  //---------------------------------------------------------------------------
  E_PROGRESS.PROGRESS_BUSY:
    _eRslt                      := StationsClearAll(TRUE); // all xts station queues clear
    IF (_eRslt = E_PROGRESS.PROGRESS_DONE)
    THEN
      _eState                   := E_PROGRESS.PROGRESS_PREPARE;
    ELSE
      IF (_eRslt = E_PROGRESS.PROGRESS_ERROR)
      THEN
        _eState                 := E_PROGRESS.PROGRESS_ERROR;
      END_IF
    END_IF

  E_PROGRESS.PROGRESS_PREPARE:
    _eRslt                      := _MoverItf[_nMover].SendToModuloPosCa(TRUE, _stMoveData);

    IF (_eRslt = E_PROGRESS.PROGRESS_ERROR)
    THEN
      _eState                   := E_PROGRESS.PROGRESS_ERROR;
      _nErrorId                 := _MoverInfo[_nMover].nErrorId;
      _eRslt                    := _MoverItf[_nMover].SendToModuloPosCa(FALSE, _stMoveData); 

    ELSIF (_eRslt = E_PROGRESS.PROGRESS_DONE)
    THEN
      _eState                   := E_PROGRESS.PROGRESS_STARTUP;
      _eRslt                    := _MoverItf[_nMover].SendToModuloPosCa(FALSE, _stMoveData);
    END_IF

  //---------------------------------------------------------------------------
  E_PROGRESS.PROGRESS_STARTUP:
    IF (_nMover > GVL_XTS.XpuInfo.nDetectedAxisCount-1)
    THEN
      // all mover are sent to start position, now prepare ticket for Mover 1
      _eState                         := E_PROGRESS.PROGRESS_CHECK;
      // ticket data
      _stMoverDataSend.nMask          := TO_USINT(EXPT(2,_StationStart.nConfiguredStopCount))-1;
      _stMoverDataSend.nMoverId       := TO_USINT(1);
      _stMoverDataSend.nTargetStation := TO_USINT(_nStartStation);
  
      IF (_nStartStation > 0) AND
         (_nStartStation < MAX_STATION+1)
      THEN
        _stListResult           := _ItfStationList[_nStartStation].AddTailValue(_stMoverDataSend); // add first mover to list of _ItfStations[_nStartStation]
      END_IF

    ELSE
      _nMover                   := _nMover + 1;                                                 // increment mover ID
      _stMoveData.rPos          := _StationStart.rPosWait + 2*_MoverItf[_nMover].RailLength;    // all other mover are commanded an extra round, to make sure that mover 1 is always leading the pack
      _eRslt                    := _MoverItf[_nMover].SendToModuloPosCa(FALSE, _stMoveData);
      _eRslt                    := _MoverItf[_nMover].SendToAbsPosCa(FALSE, _stMoveData);
      _eState                   := E_PROGRESS.PROGRESS_PREPARE;                                 // go back and trigger move
    END_IF

  //---------------------------------------------------------------------------
  E_PROGRESS.PROGRESS_CHECK:
    IF (_MoverInfo[1].bMoverInTarget)
    THEN
      IF (_GroupInfo.AllAxesStanding) // wait for all mover standstill
      THEN
        _stMoveData.rPos        := _MoverInfo[1].rAbsTargetPos;                    // Mover1 position to retrigger the movers

        IF (MAX_MOVER > 1)
        THEN
          _nMover               := 2;
          IF (_stMoveData.rPos < _MoverInfo[_nMover].rAbsActPos)
          THEN
            _stMoveData.rPos    := _stMoveData.rPos + _MoverItf[_nMover].RailLength;
          END_IF
          _eState               := E_PROGRESS.PROGRESS_OCCUPIED;
        ELSE
          _eState               := E_PROGRESS.PROGRESS_WORKING;
        END_IF
      END_IF
    END_IF

  //---------------------------------------------------------------------------
  E_PROGRESS.PROGRESS_OCCUPIED:
    _eRslt                      := _MoverItf[_nMover].SendToAbsPosCa(TRUE, _stMoveData); // retrigger

    IF (_eRslt = E_PROGRESS.PROGRESS_ERROR)
    THEN
      _eState                   := E_PROGRESS.PROGRESS_ERROR;
      _nErrorId                 := _MoverInfo[_nMover].nErrorId;
      _eRslt                    := _MoverItf[_nMover].SendToAbsPosCa(FALSE, _stMoveData); 

    ELSIF (_eRslt = E_PROGRESS.PROGRESS_DONE)
    THEN
      _eState                   := E_PROGRESS.PROGRESS_WORKING;
      _eRslt                    := _MoverItf[_nMover].SendToAbsPosCa(FALSE, _stMoveData);

      // write ticket for mover in station list
      _stMoverDataSend.nMask          := TO_USINT(EXPT(2,_StationStart.nConfiguredStopCount))-1;
      _stMoverDataSend.nMoverId       := TO_USINT(_nMover);
      _stMoverDataSend.nTargetStation := TO_USINT(_nStartStation);

      IF (_nStartStation > 0) AND
         (_nStartStation < MAX_STATION+1)
      THEN
        _stListResult                 := _ItfStationList[_nStartStation].AddTailValue(_stMoverDataSend); // enter in list
      END_IF
    END_IF

  //---------------------------------------------------------------------------
  E_PROGRESS.PROGRESS_WORKING:
    IF (_nMover > GVL_XTS.XpuInfo.nDetectedAxisCount-1)
    THEN
      _eState                   := E_PROGRESS.PROGRESS_DONE;

      IF (_eMessageLevel > E_MessageType.eMessageError)
      THEN
        _stMsg.eType            := E_MessageType.eMessageInfo;
        _stMsg.eSubdevice       := e_Subdevice.TransportUnit_General;
        _stMsg.iErrorNumber     := 0;
        _stMsg.sText            := concat( 'State: ', TO_STRING(THIS^._eState));
        _stMsg.sText            := concat(_stMsg.sText, ': ');
        _stMsg.sText            := concat(_stMsg.sText, TO_STRING(_eState));
        f_MessageSet(_stMsg);
      END_IF
    ELSE
      _nMover                   := _nMover + 1;
      IF (_stMoveData.rPos < _MoverInfo[_nMover].rAbsActPos)
      THEN
        _stMoveData.rPos        := _stMoveData.rPos + _MoverItf[_nMover].RailLength;
      END_IF
      _eState                   := E_PROGRESS.PROGRESS_OCCUPIED;
    END_IF
END_CASE
//-----------------------------------------------------------------------------
//-----------------------------------------------------------------------------

TransportStart                  := _eState;
END_METHOD

PROPERTY XpuCtrl : REFERENCE TO ST_XPU_CTRL
SET
_XpuCtrl REF= XpuCtrl;
END_SET
END_PROPERTY

PROPERTY XpuInfo : REFERENCE TO ST_XPU_INFO
SET
_XpuInfo REF= XpuInfo;
END_SET
END_PROPERTY

METHOD XpuInit : E_PROGRESS
VAR_INPUT
  Execute     : BOOL;
END_VAR
VAR_INST
  _nErrorId   : UDINT;
  _eJobReslt,
  _eState     : E_PROGRESS;
END_VAR
//-----------------------------------------------------------------------------
IF NOT Execute 
THEN 
	_eState                       := E_PROGRESS.PROGRESS_INIT; 
END_IF 
//-----------------------------------------------------------------------------
IF NOT Check() 
THEN 
	XpuInit                       := E_PROGRESS.PROGRESS_ERROR; 
	RETURN; 
END_IF
//-----------------------------------------------------------------------------
//-----------------------------------------------------------------------------
CASE _eState
OF
  E_PROGRESS.PROGRESS_INIT:
    IF Execute
    THEN
      _nErrorId                 := 0;
      _XpuCtrl.Cmd              := E_XPU_CTRL.XTS_CMD_NULL; // clear interface

      _eState                   := E_PROGRESS.PROGRESS_BUSY;
    END_IF
  //---------------------------------------------------------------------------
  //---------------------------------------------------------------------------
  E_PROGRESS.PROGRESS_BUSY:
    _XpuCtrl.Cmd                := E_XPU_CTRL.XTS_CMD_INIT; // start Xpu init

    IF (f_GetProgress(_XpuState.State) = E_PROGRESS.PROGRESS_DONE)         // check Xpu init done
    THEN
      _eState                   := E_PROGRESS.PROGRESS_PREPARE;

    ELSIF (f_GetProgress(_XpuState.State) = E_PROGRESS.PROGRESS_ERROR)     // check for error
    THEN
      _eState                   := E_PROGRESS.PROGRESS_ERROR;
    END_IF
  //---------------------------------------------------------------------------
  //---------------------------------------------------------------------------
  E_PROGRESS.PROGRESS_PREPARE:
    _XpuCtrl.Cmd                := E_XPU_CTRL.XTS_IDLE;     // Xpu start cyclic checks and mover detection

    IF (f_GetProgress(_XpuState.State) = E_PROGRESS.PROGRESS_ERROR)     // check for error
    THEN
      _eState                   := E_PROGRESS.PROGRESS_ERROR;

    ELSIF (f_GetProgress(_XpuState.State) = E_PROGRESS.PROGRESS_WORKING)      // check Xpu Idle working
    THEN
      _eState                   := E_PROGRESS.PROGRESS_STARTUP;

    END_IF
  //---------------------------------------------------------------------------
  //---------------------------------------------------------------------------
  E_PROGRESS.PROGRESS_STARTUP:
    IF (f_GetProgress(_XpuState.State) = E_PROGRESS.PROGRESS_ERROR)
    THEN
      _eState                   := E_PROGRESS.PROGRESS_ERROR;

    ELSIF (_XpuState.Check = E_XPU_CHECK.MOVER_ID_SIMULATION) OR
          (_XpuState.Check = E_XPU_CHECK.MOVER_ID_STANDARD)   OR
          (_XpuState.Check = E_XPU_CHECK.MOVER_ID_DETECTION_VALID)
    THEN
      _eState                   := E_PROGRESS.PROGRESS_DONE;

      IF (_eMessageLevel = E_MessageType.eMessageVerbose)
      THEN
        _stMsg.eType            := E_MessageType.eMessageVerbose;
        _stMsg.eSubdevice       := e_Subdevice.TransportUnit_General;
        _stMsg.iErrorNumber     := 0;
        _stMsg.sText            := concat( 'State: ', TO_STRING(THIS^._eState));
        _stMsg.sText            := concat(_stMsg.sText, ': ');
        _stMsg.sText            := concat(_stMsg.sText, TO_STRING(_eState));
        f_MessageSet(_stMsg);
      END_IF
    END_IF
END_CASE
//-----------------------------------------------------------------------------
//-----------------------------------------------------------------------------
XpuInit                         := _eState;
END_METHOD

PROPERTY XpuState : REFERENCE TO ST_XPU_STATE
SET
_XpuState ref= XpuState;
END_SET
END_PROPERTY

END_FUNCTION_BLOCK

// ---- XTS/CaGroup/FB_CaGroup.TcPOU
//---------------------------------------------------------------------------------------------------------------
//
//  HAUD 2023.12.13
//
//
//  fb_CaGroup
//  - handles CA group states
//  - add mover to group
//  - remove mover from group
//  - clear group error
//  - startup procedure for getting group ready to work
//
//
//  VAR INPUT / OUTPUT --> see properties
//
//---------------------------------------------------------------------------------------------------------------//
// This SOFTWARE is provided as an Exemple by THE PROVIDER "as is" and "with all faults." THE PROVIDER makes no  //
// representations or warranties of any kind concerning the safety, suitability, lack of viruses, inaccuracies,  //
// typographical errors, or other harmful components of this SOFTWARE. There are inherent dangers in the use of  //
// any software, and you are solely responsible for determining whether this SOFTWARE is compatible with your    //
// equipment and other software installed on your equipment. You are also solely responsible for the protection  //
// of your equipment and backup of your data, and THE PROVIDER will not be liable for any damages you may suffer //
// in connection with using, modifying, or distributing this SOFTWARE.                                           //
//---------------------------------------------------------------------------------------------------------------//
FUNCTION_BLOCK FB_CaGroup	IMPLEMENTS I_XtsTransport_CaGroup
VAR CONSTANT
{attribute 'hide'} 
  GROUP_HALT_JERK             : LREAL := 500_000.0;
{attribute 'hide'} 
  GROUP_HALT_DEC              : LREAL :=  12_500.0;
END_VAR
VAR
  _eCheck                     : E_GROUP_CHECK;
  _bError                     : BOOL;

  _GroupRef                   : REFERENCE TO Tc3_McCoordinatedMotion.AXES_GROUP_REF;

  _AxisRefMover               : REFERENCE TO ARRAY[1..MAX_MOVER] OF Tc2_MC2.AXIS_REF;
  _MoverItf                   : REFERENCE TO ARRAY[1..MAX_MOVER] OF I_XtsTransport_Mover;  // mover methods

  _stMoveData                 : ST_MOVE_DATA; // dyn constraints for _MoverItf[i].Halt(Execute, stMoveData)

  // CA group fb instances
  _fbAddAxisGroup             : ARRAY[1..MAX_MOVER] OF Tc3_McCoordinatedMotion.MC_AddAxisToGroup;
  _fbRemoveAxisGroup          : ARRAY[1..MAX_MOVER] OF Tc3_McCoordinatedMotion.MC_RemoveAxisFromGroup;

  _fbGroupDisable             : Tc3_McCoordinatedMotion.MC_GroupDisable;
  _fbGroupEnable              : Tc3_McCoordinatedMotion.MC_GroupEnable;
  _fbGroupErrorRead           : Tc3_McCoordinatedMotion.MC_GroupReadError;
  _fbGroupStatusRead          : Tc3_McCoordinatedMotion.MC_GroupReadStatus;
  _fbGroupReset               : Tc3_McCoordinatedMotion.MC_GroupReset;
  _fbGroupStop                : Tc3_McCoordinatedMotion.MC_GroupStop;

  _stGroupInfo                : ST_GROUP_INFO;  // additional bits about the state of the CA group

  _rtrigGroupStatusRead,
  _rtrigGroupErrorRead        : Tc2_Standard.R_TRIG;

  _stMsg                      : ST_Message;
  _eMessageLevel              : E_MessageType;
END_VAR

METHOD AddAll : E_PROGRESS
VAR_INPUT
  Execute     : BOOL;
END_VAR
VAR_INST
  _nErrorId   : UDINT;
  _eState     : E_PROGRESS;

  _nMover     : UINT;
END_VAR
IF NOT Execute THEN _eState     := E_PROGRESS.PROGRESS_INIT; END_IF 
IF NOT Check() THEN AddAll := E_PROGRESS.PROGRESS_ERROR; RETURN; END_IF


CASE _eState
OF
  E_PROGRESS.PROGRESS_INIT:
    IF Execute
    THEN
      _nErrorId               := 0;
      _nMover                 := 1;

      IF (_stGroupInfo.AxisCount < MAX_MOVER)
      THEN
        _eState               := E_PROGRESS.PROGRESS_BUSY;

      ELSE
        _eState               := E_PROGRESS.PROGRESS_DONE;

        IF (_eMessageLevel = E_MessageType.eMessageVerbose)
        THEN
          _stMsg.eType        := E_MessageType.eMessageVerbose;
          _stMsg.eSubdevice   := e_Subdevice.fbGroupAddAxis;
          _stMsg.iErrorNumber := _nMover;
          _stMsg.sText        := TO_STRING(_eState);
          f_MessageSet(_stMsg);
        END_IF
      END_IF
    END_IF
END_CASE
//-----------------------------------------------------------------------------
//-----------------------------------------------------------------------------
CASE _eState
OF
  E_PROGRESS.PROGRESS_BUSY:
    IF (_eMessageLevel = E_MessageType.eMessageVerbose)
    THEN
      _stMsg.eType            := E_MessageType.eMessageVerbose;
      _stMsg.eSubdevice       := e_Subdevice.fbGroupAddAxis;
      _stMsg.iErrorNumber     := _nMover;
      _stMsg.sText            := TO_STRING(_eState);
      f_MessageSet(_stMsg);
    END_IF

    _eState                   := E_PROGRESS.PROGRESS_PREPARE;
    _fbAddAxisGroup[_nMover](
                AxesGroup     := _GroupRef, 
                Axis          := _AxisRefMover[_nMover], 
                Execute       := FALSE, 
                IdentInGroup  := UDINT_TO_IDENTINGROUP(_AxisRefMover[_nMover].NcToPlc.AxisId));
END_CASE
//-----------------------------------------------------------------------------
//-----------------------------------------------------------------------------
CASE _eState
OF
  E_PROGRESS.PROGRESS_PREPARE:
    _fbAddAxisGroup[_nMover](
                AxesGroup     := _GroupRef, 
                Axis          := _AxisRefMover[_nMover], 
                Execute       := TRUE, 
                IdentInGroup  := UDINT_TO_IDENTINGROUP(_AxisRefMover[_nMover].NcToPlc.AxisId));

    IF (_fbAddAxisGroup[_nMover].Error)
    THEN
      _eState                 := E_PROGRESS.PROGRESS_ERROR;
      _nErrorId               := _fbAddAxisGroup[_nMover].ErrorId;

      _stMsg.eType            := E_MessageType.eMessageError;
      _stMsg.eSubdevice       := e_Subdevice.fbGroupAddAxis;
      _stMsg.iErrorNumber     := _nErrorId;
      _stMsg.sText            := TO_STRING(_eState);
      f_MessageSet(_stMsg);

    ELSIF (_fbAddAxisGroup[_nMover].Done)
    THEN
      _eState                 := E_PROGRESS.PROGRESS_CHECK;

      IF (_eMessageLevel = E_MessageType.eMessageVerbose)
      THEN
        _stMsg.eType          := E_MessageType.eMessageVerbose;
        _stMsg.eSubdevice     := e_Subdevice.fbGroupAddAxis;
        _stMsg.iErrorNumber   := _nMover;
        _stMsg.sText          := TO_STRING(_eState);
        f_MessageSet(_stMsg);
      END_IF
    END_IF
END_CASE
//-----------------------------------------------------------------------------
//-----------------------------------------------------------------------------
CASE _eState
OF
  E_PROGRESS.PROGRESS_CHECK:
    _eState                   := E_PROGRESS.PROGRESS_OCCUPIED;
    _fbAddAxisGroup[_nMover](
                AxesGroup     := _GroupRef, 
                Axis          := _AxisRefMover[_nMover], 
                Execute       := FALSE, 
                IdentInGroup  := UDINT_TO_IDENTINGROUP(_AxisRefMover[_nMover].NcToPlc.AxisId));
END_CASE
//-----------------------------------------------------------------------------
//-----------------------------------------------------------------------------
CASE _eState
OF
  E_PROGRESS.PROGRESS_OCCUPIED:
    IF (_nMover > MAX_MOVER-1)
    THEN
      _eState                 := E_PROGRESS.PROGRESS_DONE;

      IF (_eMessageLevel > E_MessageType.eMessageError)
      THEN
        _stMsg.eType          := E_MessageType.eMessageInfo;
        _stMsg.eSubdevice     := e_Subdevice.fbGroupAddAxis;
        _stMsg.iErrorNumber   := MAX_MOVER;
        _stMsg.sText          := TO_STRING(_eState);
        f_MessageSet(_stMsg);
      END_IF
    ELSE
      _nMover                 := _nMover + 1;
      _eState                 := E_PROGRESS.PROGRESS_BUSY;
    END_IF
END_CASE
//-----------------------------------------------------------------------------
//-----------------------------------------------------------------------------

AddAll                   := _eState;
END_METHOD

PROPERTY AxisRef : REFERENCE TO ARRAY[1..MAX_MOVER] OF Tc2_MC2.AXIS_REF
SET
_AxisRefMover REF= AxisRef;
END_SET
END_PROPERTY

METHOD PROTECTED Check : BOOL

IF NOT __ISVALIDREF(_GroupRef)
THEN
  _eCheck                     := E_GROUP_CHECK.CHECK_GROUP_REF_INVALID;
  RETURN;
END_IF

IF NOT __ISVALIDREF(_AxisRefMover)
THEN
  _eCheck                     := E_GROUP_CHECK.CHECK_AXIS_REF_INVALID;
  RETURN;
END_IF

IF NOT __ISVALIDREF(_MoverItf)
THEN
  _eCheck                     := E_GROUP_CHECK.CHECK_Mover_ITF_REF_INVALID;
  RETURN;
END_IF

_eCheck                       := E_GROUP_CHECK.CHECK_DONE;
Check                         := TRUE;
END_METHOD

METHOD Disable : E_PROGRESS
VAR_INPUT
  Execute     : BOOL;
END_VAR
VAR_INST
  _nErrorId   : UDINT;
  _eState     : E_PROGRESS;

  _nMover     : UINT;
END_VAR
IF NOT Execute THEN _eState       := E_PROGRESS.PROGRESS_INIT; END_IF 
IF NOT Check() THEN Disable  := E_PROGRESS.PROGRESS_ERROR; RETURN; END_IF


CASE _eState
OF
  E_PROGRESS.PROGRESS_INIT:
    IF Execute
    THEN
      _nErrorId               := 0;
      _nMover                 := 1;
      _eState                 := E_PROGRESS.PROGRESS_BUSY;
    END_IF
END_CASE
//-----------------------------------------------------------------------------
//-----------------------------------------------------------------------------
CASE _eState
OF
  E_PROGRESS.PROGRESS_BUSY:
    IF (_stGroupInfo.CaGroupState = E_CA_GROUP_STATE.mcGroupStateDisabled)
    THEN
      _eState                 := E_PROGRESS.PROGRESS_DONE;

      IF (_eMessageLevel = E_MessageType.eMessageVerbose)
      THEN
        _stMsg.eType          := E_MessageType.eMessageVerbose;
        _stMsg.eSubdevice     := e_Subdevice.fbGroupDisable;
        _stMsg.iErrorNumber   := _nErrorId;
        _stMsg.sText          := TO_STRING(_eState);
        f_MessageSet(_stMsg);
      END_IF
    ELSE
      _eState                 := E_PROGRESS.PROGRESS_PREPARE;
      _fbGroupDisable(
                AxesGroup     := _GroupRef, 
                Execute       := FALSE);

      _fbGroupReset(
                AxesGroup     := _GroupRef, 
                Execute       := FALSE);
  
      IF (_eMessageLevel = E_MessageType.eMessageVerbose)
      THEN
        _stMsg.eType          := E_MessageType.eMessageVerbose;
        _stMsg.eSubdevice     := e_Subdevice.fbGroupDisable;
        _stMsg.iErrorNumber   := _nErrorId;
        _stMsg.sText          := TO_STRING(_eState);
        f_MessageSet(_stMsg);
      END_IF
    END_IF
END_CASE
//-----------------------------------------------------------------------------
//-----------------------------------------------------------------------------
CASE _eState
OF
  E_PROGRESS.PROGRESS_PREPARE:
    _fbGroupReset(
                AxesGroup     := _GroupRef, 
                Execute       := TRUE);

    IF (_fbGroupReset.Error)
    THEN
      _eState                 := E_PROGRESS.PROGRESS_ERROR;
      _nErrorId               := _fbGroupReset.ErrorId;

      _stMsg.eType            := E_MessageType.eMessageError;
      _stMsg.eSubdevice       := e_Subdevice.fbGroupReset;
      _stMsg.iErrorNumber     := _nErrorId;
      _stMsg.sText            := TO_STRING(_eState);
      f_MessageSet(_stMsg);

      _fbGroupReset(
                AxesGroup     := _GroupRef, 
                Execute       := FALSE);
    ELSE
      IF (_fbGroupReset.Done)
      THEN
        _eState               := E_PROGRESS.PROGRESS_STARTUP;
        _fbGroupReset(
                AxesGroup     := _GroupRef, 
                Execute       := FALSE);
      END_IF
    END_IF
END_CASE
//-----------------------------------------------------------------------------
//-----------------------------------------------------------------------------
CASE _eState
OF
  E_PROGRESS.PROGRESS_STARTUP:
    _fbGroupDisable(
              AxesGroup       := _GroupRef, 
              Execute         := TRUE); 

    IF (_fbGroupDisable.Error)
    THEN
      _eState                 := E_PROGRESS.PROGRESS_ERROR;
      _nErrorId               := _fbGroupDisable.ErrorId;

      _stMsg.eType            := E_MessageType.eMessageError;
      _stMsg.eSubdevice       := e_Subdevice.fbGroupDisable;
      _stMsg.iErrorNumber     := _nErrorId;
      _stMsg.sText            := TO_STRING(_eState);
      f_MessageSet(_stMsg);

      _fbGroupDisable(
              AxesGroup       := _GroupRef, 
              Execute         := FALSE); 


    ELSIF (_fbGroupDisable.Done)
    THEN
      _eState                 := E_PROGRESS.PROGRESS_DONE;

      IF (_eMessageLevel > E_MessageType.eMessageError)
      THEN
        _stMsg.eType          := E_MessageType.eMessageInfo;
        _stMsg.eSubdevice     := e_Subdevice.fbGroupDisable;
        _stMsg.iErrorNumber   := _nErrorId;
        _stMsg.sText          := TO_STRING(_eState);
        f_MessageSet(_stMsg);
      END_IF

      _fbGroupDisable(
              AxesGroup       := _GroupRef, 
              Execute         := FALSE); 
    END_IF
END_CASE
//-----------------------------------------------------------------------------
//-----------------------------------------------------------------------------

Disable                  := _eState;
END_METHOD

METHOD Enable : E_PROGRESS
VAR_INPUT
  Execute     : BOOL;
END_VAR
VAR_INST
  _nErrorId   : UDINT;
  _eState     : E_PROGRESS;

  _nMover     : UINT;
END_VAR
IF NOT Execute THEN _eState       := E_PROGRESS.PROGRESS_INIT; END_IF 
IF NOT Check() THEN Enable   := E_PROGRESS.PROGRESS_ERROR; RETURN; END_IF


CASE _eState
OF
  E_PROGRESS.PROGRESS_INIT:
    IF Execute
    THEN
      _nErrorId               := 0;
      _nMover                 := 1;
      _eState                 := E_PROGRESS.PROGRESS_BUSY;
    END_IF
END_CASE
//-----------------------------------------------------------------------------
//-----------------------------------------------------------------------------
CASE _eState
OF
  E_PROGRESS.PROGRESS_BUSY:
    _eState                   := E_PROGRESS.PROGRESS_PREPARE;
    _fbGroupEnable(
                AxesGroup     := _GroupRef, 
                Execute       := FALSE);

    IF (_eMessageLevel = E_MessageType.eMessageVerbose)
    THEN
      _stMsg.eType            := E_MessageType.eMessageVerbose;
      _stMsg.eSubdevice       := e_Subdevice.fbGroupEnable;
      _stMsg.iErrorNumber     := _nErrorId;
      _stMsg.sText            := TO_STRING(_eState);
      f_MessageSet(_stMsg);
    END_IF
END_CASE
//-----------------------------------------------------------------------------
//-----------------------------------------------------------------------------
CASE _eState
OF
  E_PROGRESS.PROGRESS_PREPARE:
    _fbGroupEnable(
                AxesGroup     := _GroupRef, 
                Execute       := TRUE);

    IF (_fbGroupEnable.Error)
    THEN
      _eState                 := E_PROGRESS.PROGRESS_ERROR;
      _nErrorId               := _fbGroupEnable.ErrorId;

      _stMsg.eType            := E_MessageType.eMessageError;
      _stMsg.eSubdevice       := e_Subdevice.fbGroupEnable;
      _stMsg.iErrorNumber     := _nErrorId;
      _stMsg.sText            := TO_STRING(_eState);
      f_MessageSet(_stMsg);

      _fbGroupEnable(
                AxesGroup     := _GroupRef, 
                Execute       := FALSE);

    ELSIF (_fbGroupEnable.Done)
    THEN
      _eState                 := E_PROGRESS.PROGRESS_DONE;

      IF (_eMessageLevel > E_MessageType.eMessageError)
      THEN
        _stMsg.eType          := E_MessageType.eMessageInfo;
        _stMsg.eSubdevice     := e_Subdevice.fbGroupEnable;
        _stMsg.iErrorNumber   := _nErrorId;
        _stMsg.sText          := TO_STRING(_eState);
        f_MessageSet(_stMsg);
      END_IF
      _fbGroupEnable(
                AxesGroup     := _GroupRef, 
                Execute       := FALSE);
    END_IF
END_CASE
//-----------------------------------------------------------------------------
//-----------------------------------------------------------------------------

Enable                   := _eState;
END_METHOD

PROPERTY GroupInfo : reference to ST_GROUP_INFO
GET
GroupInfo REF= _stGroupInfo;
END_GET
END_PROPERTY

PROPERTY GroupRef : reference to Tc3_McCoordinatedMotion.AXES_GROUP_REF
GET
GroupRef REF= _GroupRef;
END_GET
SET
_GroupRef REF= GroupRef;
END_SET
END_PROPERTY

METHOD InfoCycle : DWORD
VAR_INPUT
  EnableCycle          : BOOL;
END_VAR
VAR_INST
  _nErrorIdADS,
  _nErrorIdRead   : UDINT;

  _nIdx           : udint;
END_VAR
IF NOT Check() THEN RETURN; END_IF

_stMsg.eDevice                              := e_Device.CaGroup;

//-----------------------------------------------------------------------------------------------
// cyclic CA group
//-----------------------------------------------------------------------------------------------
_fbGroupStatusRead(
              AxesGroup                     := _GroupRef, 
              Enable                        := EnableCycle, 
              Valid                         => _stGroupInfo.GroupStatusValid, 
              Busy                          => _stGroupInfo.GroupStatusBusy, 
              GroupMoving                   => _stGroupInfo.GroupMoving, 
              GroupHoming                   => _stGroupInfo.GroupHoming, 
              GroupErrorStop                => _stGroupInfo.GroupErrorStop, 
              GroupNotReady                 => _stGroupInfo.GroupNotReady, 
              GroupStandby                  => _stGroupInfo.GroupStandby, 
              GroupStopping                 => _stGroupInfo.GroupStopping, 
              GroupDisabled                 => _stGroupInfo.GroupDisabled, 
              AllAxesStanding               => _stGroupInfo.AllAxesStanding, 
              ConstantVelocity              => _stGroupInfo.ConstantVelocity, 
              Accelerating                  => _stGroupInfo.Accelerating, 
              Decelerating                  => _stGroupInfo.Decelerating, 
              InPosition                    => _stGroupInfo.InPosition, 
              Error                         => _stGroupInfo.GroupError, 
              ErrorId                       => );

_fbGroupErrorRead(
              AxesGroup                     := _GroupRef, 
              Enable                        := EnableCycle, 
              ErrorId                       => , 
              GroupErrorId                  => _stGroupInfo.GroupErrorId);


_stGroupInfo.AxisCount                      := _GroupRef.NcToPlc.CA.Common.GroupAxesCount;
_stGroupInfo.CaGroupOID                     := _GroupRef.NcToPlc.CA.Common.GroupOID;
_stGroupInfo.CaGroupState                   := TO_UINT(_GroupRef.NcToPlc.CA.Common.GroupStatus.State);

_stGroupInfo.AxisCountEnabled               := 0;
FOR _nIdx := 1 TO MAX_MOVER
DO
  IF (_AxisRefMover[_nIdx].Status.ControlLoopClosed)
  THEN
    _stGroupInfo.AxisCountEnabled           := _stGroupInfo.AxisCountEnabled + 1;
  END_IF
END_FOR	
			  
// fetch internal fb error
_rtrigGroupErrorRead(CLK                    := _fbGroupErrorRead.Error);
IF _rtrigGroupErrorRead.Q
THEN
  _nErrorIdADS                              := _fbGroupErrorRead.ErrorId;

  _stMsg.eType                              := E_MessageType.eMessageError;
  _stMsg.eSubdevice                         := e_Subdevice.fbGroupErrorRead;
  _stMsg.iErrorNumber                       := _nErrorIdADS;
  _stMsg.sText                              := '';
  f_MessageSet(_stMsg);
END_IF

// Dyn constrainst for McHaltAll(method)
_stMoveData.rJerk                           := GROUP_HALT_JERK;
_stMoveData.rAcc                            := GROUP_HALT_DEC;
END_METHOD

METHOD McHaltAll : E_PROGRESS
VAR_INPUT
  Execute       : BOOL;
END_VAR
VAR_INST
  _nErrorId     : UDINT;
  _eState       : E_PROGRESS;
  _eResult      : E_PROGRESS;

  _nMover       : UINT;

  _nRepeat      : UINT;
END_VAR
IF NOT Execute 
THEN 
	_eState     := E_PROGRESS.PROGRESS_INIT; 
END_IF 
IF NOT Check() 
THEN 
	McHaltAll   := E_PROGRESS.PROGRESS_ERROR; 
	RETURN; 
END_IF


CASE _eState
OF
  E_PROGRESS.PROGRESS_INIT:
    IF Execute
    THEN
      _fbGroupStop(
              AxesGroup       := _GroupRef, 
              Execute         := FALSE, 
              Deceleration    := GROUP_HALT_DEC, 
              Jerk            := GROUP_HALT_JERK);

      _nErrorId               := 0;
      _nMover                 := 1;
      _eState                 := E_PROGRESS.PROGRESS_BUSY;
    END_IF
END_CASE

//-----------------------------------------------------------------------------
//-----------------------------------------------------------------------------
CASE _eState
OF
  E_PROGRESS.PROGRESS_BUSY:
    IF NOT (_stGroupInfo.CaGroupState = E_CA_GROUP_STATE.mcGroupStateMoving)
    THEN
      _eState                   := E_PROGRESS.PROGRESS_PREPARE;
    ELSE
      _fbGroupStop(
                AxesGroup       := _GroupRef, 
                Execute         := TRUE, 
                Deceleration    := GROUP_HALT_DEC, 
                Jerk            := GROUP_HALT_JERK);
  
      IF (_fbGroupStop.Error)
      THEN
        _stMsg.eType            := E_MessageType.eMessageError;
        _stMsg.eSubdevice       := e_Subdevice.fbGroupStop;
        _stMsg.iErrorNumber     := _fbGroupStop.ErrorId;
        _stMsg.sText            := TO_STRING(_eState);
        f_MessageSet(_stMsg);
  
        _nRepeat                := _nRepeat + 1;
        _eState                 := E_PROGRESS.PROGRESS_PREPARE;
      ELSE
        IF (_fbGroupStop.Done)
        THEN
          IF (_eMessageLevel = E_MessageType.eMessageVerbose)
          THEN
            _stMsg.eType        := E_MessageType.eMessageVerbose;
            _stMsg.eSubdevice   := e_Subdevice.fbGroupStop;
            _stMsg.iErrorNumber := MAX_MOVER;
            _stMsg.sText        := TO_STRING(_eState);
            f_MessageSet(_stMsg);
          END_IF
          _nRepeat              := 0;
          _eState               := E_PROGRESS.PROGRESS_PREPARE;
        END_IF
      END_IF
    END_IF
END_CASE

//-----------------------------------------------------------------------------
//-----------------------------------------------------------------------------
CASE _eState
OF
  E_PROGRESS.PROGRESS_PREPARE:
    _eState                   := E_PROGRESS.PROGRESS_WORKING;
    _fbGroupStop(
              AxesGroup       := _GroupRef, 
              Execute         := FALSE, 
              Deceleration    := GROUP_HALT_DEC, 
              Jerk            := GROUP_HALT_JERK);

    _eResult                  := _MoverItf[_nMover].Reset(FALSE);
    _eResult                  := _MoverItf[_nMover].Halt(FALSE, _stMoveData);
END_CASE
//-----------------------------------------------------------------------------
//-----------------------------------------------------------------------------
CASE _eState
OF
  E_PROGRESS.PROGRESS_WORKING:
    _eResult                  := _MoverItf[_nMover].Halt(TRUE, _stMoveData);

    IF (_eResult = E_PROGRESS.PROGRESS_DONE)
    THEN
      _eResult                := _MoverItf[_nMover].Halt(FALSE, _stMoveData);
      _eState                 := E_PROGRESS.PROGRESS_STARTUP;

    ELSIF (_eResult = E_PROGRESS.PROGRESS_ERROR)
    THEN
      _nErrorId               := _AxisRefMover[_nMover].NcToPlc.ErrorCode;
      _MoverItf[_nMover].Reset(TRUE);

      _stMsg.eType            := E_MessageType.eMessageError;
      _stMsg.eSubdevice       := e_Subdevice.fbHalt;
      _stMsg.iErrorNumber     := _nErrorId;
      _stMsg.sText            := concat( 'McHaltAll: ', TO_STRING(_eResult));
      _stMsg.sText            := concat(_stMsg.sText, ' MoverId: ');
      _stMsg.sText            := concat(_stMsg.sText, TO_STRING(_nMover));
      f_MessageSet(_stMsg);

      _eState                 := E_PROGRESS.PROGRESS_PREPARE;
    END_IF
END_CASE

//-----------------------------------------------------------------------------
//-----------------------------------------------------------------------------
CASE _eState
OF
  E_PROGRESS.PROGRESS_STARTUP:
    IF (_nMover > MAX_MOVER-1)
    THEN
      _eState                 := E_PROGRESS.PROGRESS_CHECK;
    ELSE
      _nMover                 := _nMover + 1;
      _eState                 := E_PROGRESS.PROGRESS_PREPARE;
    END_IF
END_CASE

//-----------------------------------------------------------------------------
//-----------------------------------------------------------------------------
CASE _eState
OF
  E_PROGRESS.PROGRESS_CHECK:
    _eState                   := E_PROGRESS.PROGRESS_DONE;

    IF (_eMessageLevel > E_MessageType.eMessageError)
    THEN
      _stMsg.eType            := E_MessageType.eMessageInfo;
      _stMsg.eSubdevice       := e_Subdevice.fbCaGroup;
      _stMsg.iErrorNumber     := MAX_MOVER;
      _stMsg.sText            := concat('McHaltAll: ', TO_STRING(_eState));
      f_MessageSet(_stMsg);
    END_IF
END_CASE
//-----------------------------------------------------------------------------
//-----------------------------------------------------------------------------
McHaltAll                     := _eState;
END_METHOD

METHOD McResetAll : E_PROGRESS
VAR_INPUT
  Execute       : BOOL;
END_VAR
VAR_INST
  _nErrorId     : UDINT;
  _eRslt,
  _eState       : E_PROGRESS;

  _nMover       : UINT;
END_VAR
IF NOT Execute THEN _eState     := E_PROGRESS.PROGRESS_INIT; END_IF 
IF NOT Check() THEN McResetAll  := E_PROGRESS.PROGRESS_ERROR; RETURN; END_IF


//-----------------------------------------------------------------------------
//-----------------------------------------------------------------------------
CASE _eState
OF
  E_PROGRESS.PROGRESS_INIT:
    IF Execute
    THEN
      _nErrorId                 := 0;
      _nMover                   := 1;

      _eState                   := E_PROGRESS.PROGRESS_BUSY;
    END_IF
END_CASE
//-----------------------------------------------------------------------------
//-----------------------------------------------------------------------------
CASE _eState
OF
  E_PROGRESS.PROGRESS_BUSY:
    _eState                     := E_PROGRESS.PROGRESS_PREPARE;
    _eRslt                      := _MoverItf[_nMover].Reset(FALSE);
END_CASE
//-----------------------------------------------------------------------------
//-----------------------------------------------------------------------------
CASE _eState
OF
  E_PROGRESS.PROGRESS_PREPARE:
    _eRslt                      := _MoverItf[_nMover].Reset(TRUE);

    IF (_eRslt = E_PROGRESS.PROGRESS_ERROR)
    THEN
      _eState                   := E_PROGRESS.PROGRESS_BUSY;

    ELSIF (_eRslt = E_PROGRESS.PROGRESS_DONE)
    THEN
      _eState                   := E_PROGRESS.PROGRESS_STARTUP;
    END_IF
END_CASE
//-----------------------------------------------------------------------------
//-----------------------------------------------------------------------------
CASE _eState
OF
  E_PROGRESS.PROGRESS_STARTUP:
    _eState                     := E_PROGRESS.PROGRESS_CHECK;
    _eRslt                      := _MoverItf[_nMover].Reset(FALSE);
END_CASE
//-----------------------------------------------------------------------------
//-----------------------------------------------------------------------------
CASE _eState
OF
  E_PROGRESS.PROGRESS_CHECK:
    IF (_nMover > MAX_MOVER-1)
    THEN
      _eState                   := E_PROGRESS.PROGRESS_DONE;

      IF (_eMessageLevel = E_MessageType.eMessageVerbose)
      THEN
        _stMsg.eType            := E_MessageType.eMessageVerbose;
        _stMsg.eSubdevice       := e_Subdevice.fbReset;
        _stMsg.iErrorNumber     := 0;
        _stMsg.sText            := concat( 'State: ', TO_STRING(_eState));
        f_MessageSet(_stMsg);
      END_IF
    ELSE
      _nMover                   := _nMover + 1;
      _eState                   := E_PROGRESS.PROGRESS_BUSY;
    END_IF
END_CASE
//-----------------------------------------------------------------------------
//-----------------------------------------------------------------------------


McResetAll                      := _eState;
END_METHOD

PROPERTY MessageLevel : e_messagetype
SET
_eMessageLevel := MessageLevel;
END_SET
END_PROPERTY

PROPERTY MoverItf : reference TO ARRAY[1..MAX_MOVER] OF I_XtsTransport_Mover
SET
_MoverItf REF= MoverItf;
END_SET
END_PROPERTY

METHOD RemoveAll : E_PROGRESS
VAR_INPUT
  Execute     : BOOL;
END_VAR
VAR_INST
  _nErrorId   : UDINT;
  _eState     : E_PROGRESS;

  _nMover     : UINT;
END_VAR
IF NOT Execute THEN _eState         := E_PROGRESS.PROGRESS_INIT; END_IF 
IF NOT Check() THEN RemoveAll  := E_PROGRESS.PROGRESS_ERROR; RETURN; END_IF


CASE _eState
OF
  E_PROGRESS.PROGRESS_INIT:
    IF Execute
    THEN
      _nErrorId               := 0;
      _nMover                 := 1;

      IF (_stGroupInfo.AxisCount > 0)
      THEN
        _eState               := E_PROGRESS.PROGRESS_BUSY;
      ELSE
        _eState               := E_PROGRESS.PROGRESS_DONE;

        IF (_eMessageLevel = E_MessageType.eMessageVerbose)
        THEN
          _stMsg.eType        := E_MessageType.eMessageVerbose;
          _stMsg.eSubdevice   := e_Subdevice.fbGroupRemoveAxis;
          _stMsg.iErrorNumber := _stGroupInfo.AxisCount;
          _stMsg.sText        := TO_STRING(_eState);
          f_MessageSet(_stMsg);
        END_IF
      END_IF
    END_IF
END_CASE
//-----------------------------------------------------------------------------
//-----------------------------------------------------------------------------
CASE _eState
OF
  E_PROGRESS.PROGRESS_BUSY:
    IF (_eMessageLevel = E_MessageType.eMessageVerbose)
    THEN
      _stMsg.eType          := E_MessageType.eMessageVerbose;
      _stMsg.eSubdevice     := e_Subdevice.fbGroupRemoveAxis;
      _stMsg.iErrorNumber   := _nMover;
      _stMsg.sText          := TO_STRING(_eState);
      //f_MessageSet(_stMsg);
    END_IF

    _eState                 := E_PROGRESS.PROGRESS_PREPARE;
    _fbRemoveAxisGroup[_nMover](
            AxesGroup       := _GroupRef, 
            Execute         := FALSE,
            IdentInGroup    := UDINT_TO_IDENTINGROUP(_AxisRefMover[_nMover].NcToPlc.AxisId));
END_CASE
//-----------------------------------------------------------------------------
//-----------------------------------------------------------------------------
CASE _eState
OF
  E_PROGRESS.PROGRESS_PREPARE:
    _fbRemoveAxisGroup[_nMover](
              AxesGroup       := _GroupRef, 
              Execute         := TRUE,
              IdentInGroup    := UDINT_TO_IDENTINGROUP(_AxisRefMover[_nMover].NcToPlc.AxisId));

    IF (_fbRemoveAxisGroup[_nMover].Error)
    THEN
      _eState                 := E_PROGRESS.PROGRESS_ERROR;
      _nErrorId               := _fbRemoveAxisGroup[_nMover].ErrorId;

      _stMsg.eType            := E_MessageType.eMessageError;
      _stMsg.eSubdevice       := e_Subdevice.fbGroupRemoveAxis;
      _stMsg.iErrorNumber     := _nErrorId;
      _stMsg.sText            := TO_STRING(_eState);
      f_MessageSet(_stMsg);

    ELSIF (_fbRemoveAxisGroup[_nMover].Done)
    THEN
      _eState                 := E_PROGRESS.PROGRESS_CHECK;

      IF (_eMessageLevel = E_MessageType.eMessageVerbose)
      THEN
        _stMsg.eType          := E_MessageType.eMessageVerbose;
        _stMsg.eSubdevice     := e_Subdevice.fbGroupRemoveAxis;
        _stMsg.iErrorNumber   := _nMover;
        _stMsg.sText          := TO_STRING('DONE');
        //f_MessageSet(_stMsg);
      END_IF
    END_IF
END_CASE
//-----------------------------------------------------------------------------
//-----------------------------------------------------------------------------
CASE _eState
OF
  E_PROGRESS.PROGRESS_CHECK:
    _eState                   := E_PROGRESS.PROGRESS_OCCUPIED;
    _fbRemoveAxisGroup[_nMover](
              AxesGroup       := _GroupRef, 
              Execute         := FALSE,
              IdentInGroup    := UDINT_TO_IDENTINGROUP(_AxisRefMover[_nMover].NcToPlc.AxisId));
END_CASE
//-----------------------------------------------------------------------------
//-----------------------------------------------------------------------------
CASE _eState
OF
  E_PROGRESS.PROGRESS_OCCUPIED:
    IF (_nMover > MAX_MOVER-1)
    THEN
      _eState                 := E_PROGRESS.PROGRESS_DONE;

      IF (_eMessageLevel > E_MessageType.eMessageError)
      THEN
        _stMsg.eType          := E_MessageType.eMessageInfo;
        _stMsg.eSubdevice     := e_Subdevice.fbGroupRemoveAxis;
        _stMsg.iErrorNumber   := MAX_MOVER;
        _stMsg.sText          := TO_STRING(_eState);
        f_MessageSet(_stMsg);
      END_IF
    ELSE
      _nMover                 := _nMover + 1;
      _eState                 := E_PROGRESS.PROGRESS_BUSY;
    END_IF
END_CASE
//-----------------------------------------------------------------------------
//-----------------------------------------------------------------------------

RemoveAll                := _eState;
END_METHOD

METHOD Reset : E_PROGRESS
VAR_INPUT
  Execute     : BOOL;
END_VAR
VAR_INST
  _nErrorId   : UDINT;
  _eState     : E_PROGRESS;

  _nMover     : UINT;
END_VAR
IF NOT Execute 
THEN 
	_eState := E_PROGRESS.PROGRESS_INIT; 
END_IF 
IF NOT Check() 
THEN 
	Reset := E_PROGRESS.PROGRESS_ERROR; 
	RETURN; 
END_IF


CASE _eState
OF
  E_PROGRESS.PROGRESS_INIT:
    IF Execute
    THEN
      _nErrorId                 := 0;
      _nMover                   := 1;
      _stGroupInfo.GroupErrorId := 0;
      _stGroupInfo.GroupError   := FALSE;

      _eState                   := E_PROGRESS.PROGRESS_BUSY;
    END_IF
END_CASE
//-----------------------------------------------------------------------------
//-----------------------------------------------------------------------------
CASE _eState
OF
  E_PROGRESS.PROGRESS_BUSY:
    _eState                     := E_PROGRESS.PROGRESS_PREPARE;
    _fbGroupReset(
              AxesGroup         := _GroupRef, 
              Execute           := FALSE);

    IF (_eMessageLevel = E_MessageType.eMessageVerbose)
    THEN
      _stMsg.eType              := E_MessageType.eMessageVerbose;
      _stMsg.eSubdevice         := e_Subdevice.fbGroupReset;
      _stMsg.iErrorNumber       := 0;
      _stMsg.sText              := TO_STRING(_eState);
      //f_MessageSet(_stMsg);
    END_IF
END_CASE
//-----------------------------------------------------------------------------
//-----------------------------------------------------------------------------
CASE _eState
OF
  E_PROGRESS.PROGRESS_PREPARE:
    _fbGroupReset(
              AxesGroup         := _GroupRef, 
              Execute           := TRUE);

    IF (_fbGroupReset.Error)
    THEN
      _eState                   := E_PROGRESS.PROGRESS_ERROR;
      _nErrorId                 := _fbGroupReset.ErrorId;

      _stMsg.eType              := E_MessageType.eMessageError;
      _stMsg.eSubdevice         := e_Subdevice.fbGroupReset;
      _stMsg.iErrorNumber       := _nErrorId;
      _stMsg.sText              := TO_STRING(_eState);
      f_MessageSet(_stMsg);

      _fbGroupReset(
              AxesGroup         := _GroupRef, 
              Execute           := FALSE); 

    ELSIF (_fbGroupReset.Done)
    THEN
      _eState                   := E_PROGRESS.PROGRESS_DONE;

      IF (_eMessageLevel > E_MessageType.eMessageError)
      THEN
        _stMsg.eType            := E_MessageType.eMessageInfo;
        _stMsg.eSubdevice       := e_Subdevice.fbGroupReset;
        _stMsg.iErrorNumber     := _nErrorId;
        _stMsg.sText            := TO_STRING(_eState);
        f_MessageSet(_stMsg);
      END_IF

      _fbGroupReset(
              AxesGroup         := _GroupRef, 
              Execute           := FALSE); 
    END_IF
END_CASE
//-----------------------------------------------------------------------------
//-----------------------------------------------------------------------------

Reset                           := _eState;
END_METHOD

METHOD Stop : E_PROGRESS
VAR_INPUT
  Execute     : BOOL;
END_VAR
VAR_INST
  _nErrorId   : UDINT;
  _eState     : E_PROGRESS;

  _nMover     : UINT;
  _nRepeat    : uint;
END_VAR
IF NOT Execute 
THEN 
	_eState := E_PROGRESS.PROGRESS_INIT; 
END_IF 
IF NOT Check() 
THEN 
	Stop := E_PROGRESS.PROGRESS_ERROR; 
	RETURN; 
END_IF


CASE _eState
OF
  E_PROGRESS.PROGRESS_INIT:
    IF Execute
    THEN
      _nRepeat                  := 0;
      _nErrorId                 := 0;
      _nMover                   := 1;
      _eState                   := E_PROGRESS.PROGRESS_BUSY;
    END_IF
END_CASE
//-----------------------------------------------------------------------------
//-----------------------------------------------------------------------------
CASE _eState
OF
  E_PROGRESS.PROGRESS_BUSY:
    _eState                     := E_PROGRESS.PROGRESS_PREPARE;
    _fbGroupStop(
                AxesGroup       := _GroupRef, 
                Execute         := FALSE, 
                Deceleration    := GROUP_HALT_DEC, 
                Jerk            := GROUP_HALT_JERK);

    IF (_eMessageLevel = E_MessageType.eMessageVerbose)
    THEN
      _stMsg.eType              := E_MessageType.eMessageVerbose;
      _stMsg.eSubdevice         := e_Subdevice.fbGroupStop;
      _stMsg.iErrorNumber       := 0;
      _stMsg.sText              := TO_STRING(_eState);
      f_MessageSet(_stMsg);
    END_IF
END_CASE
//-----------------------------------------------------------------------------
//-----------------------------------------------------------------------------
CASE _eState
OF
  E_PROGRESS.PROGRESS_PREPARE:
    _fbGroupStop(
                AxesGroup       := _GroupRef, 
                Execute         := TRUE, 
                Deceleration    := GROUP_HALT_DEC, 
                Jerk            := GROUP_HALT_JERK);

    IF (_fbGroupStop.Error)
    THEN
      _eState                   := E_PROGRESS.PROGRESS_STARTUP;
      _nErrorId                 := _fbGroupStop.ErrorId;

      _stMsg.eType              := E_MessageType.eMessageError;
      _stMsg.eSubdevice         := e_Subdevice.fbGroupStop;
      _stMsg.iErrorNumber       := _nErrorId;
      _stMsg.sText              := TO_STRING(_eState);
      f_MessageSet(_stMsg);

      _fbGroupReset(
              AxesGroup         := _GroupRef, 
              Execute           := FALSE); 

    ELSIF (_fbGroupStop.Done)
    THEN
      _eState                   := E_PROGRESS.PROGRESS_DONE;

      IF (_eMessageLevel > E_MessageType.eMessageError)
      THEN
        _stMsg.eType            := E_MessageType.eMessageInfo;
        _stMsg.eSubdevice       := e_Subdevice.fbGroupStop;
        _stMsg.iErrorNumber     := _nErrorId;
        _stMsg.sText            := TO_STRING(_eState);
        f_MessageSet(_stMsg);
      END_IF

      _fbGroupStop(
                AxesGroup       := _GroupRef, 
                Execute         := FALSE, 
                Deceleration    := GROUP_HALT_DEC, 
                Jerk            := GROUP_HALT_JERK);
    END_IF
END_CASE
//-----------------------------------------------------------------------------
//-----------------------------------------------------------------------------
CASE _eState
OF
  E_PROGRESS.PROGRESS_STARTUP:
    _fbGroupReset(
              AxesGroup         := _GroupRef, 
              Execute           := TRUE);

    IF (_fbGroupReset.Error)
    THEN
      _nRepeat                  := _nRepeat + 1;
      IF (_nRepeat > 2)
      THEN
        _eState                 := E_PROGRESS.PROGRESS_ERROR;
      END_IF
      _nErrorId                 := _fbGroupReset.ErrorId;

      _stMsg.eType              := E_MessageType.eMessageError;
      _stMsg.eSubdevice         := e_Subdevice.fbGroupStop;
      _stMsg.iErrorNumber       := _nErrorId;
      _stMsg.sText              := TO_STRING(_eState);
      f_MessageSet(_stMsg);

      _fbGroupReset(
              AxesGroup         := _GroupRef, 
              Execute           := FALSE); 

    ELSIF (_fbGroupReset.Done)
    THEN
      _eState                   := E_PROGRESS.PROGRESS_BUSY;

      IF (_eMessageLevel > E_MessageType.eMessageError)
      THEN
        _stMsg.eType            := E_MessageType.eMessageInfo;
        _stMsg.eSubdevice       := e_Subdevice.fbGroupStop;
        _stMsg.iErrorNumber     := _nErrorId;
        _stMsg.sText            := TO_STRING(_eState);
        f_MessageSet(_stMsg);
      END_IF

      _fbGroupReset(
              AxesGroup         := _GroupRef, 
              Execute           := FALSE); 
    END_IF
END_CASE
//-----------------------------------------------------------------------------
//-----------------------------------------------------------------------------

Stop                            := _eState;
END_METHOD

END_FUNCTION_BLOCK

// ---- XTS/Mover/fb_MoverCtrl.TcPOU
//---------------------------------------------------------------------------------------------------------------
//
//  HAUD 2023.12.18
//
//  - XTS_TRANSPORT_LAYER
//
//  fb_MoverCtrl
//  - accepts orders (E_MOVER_CTRL) via cyclic struct interface to execute
//  - interface struct  to extern control
//
//
//---------------------------------------------------------------------------------------------------------------
// This SOFTWARE is provided as an Exemple by THE PROVIDER "as is" and "with all faults." THE PROVIDER makes no 
// representations or warranties of any kind concerning the safety, suitability, lack of viruses, inaccuracies, 
// typographical errors, or other harmful components of this SOFTWARE. There are inherent dangers in the use of 
// any software, and you are solely responsible for determining whether this SOFTWARE is compatible with your 
// equipment and other software installed on your equipment. You are also solely responsible for the protection 
// of your equipment and backup of your data, and THE PROVIDER will not be liable for any damages you may suffer 
// in connection with using, modifying, or distributing this SOFTWARE.
//---------------------------------------------------------------------------------------------------------------
FUNCTION_BLOCK fb_MoverCtrl EXTENDS fb_Mover
VAR
  // Ctrl and State for executing commands
  _stCtrl           : REFERENCE TO ARRAY[1..MAX_MOVER] OF ST_MOVER_CTRL;
  _stState          : REFERENCE TO ARRAY[1..MAX_MOVER] OF ST_MOVER_STATE;

  // data structures to use with commands
  _stMoveData       : REFERENCE TO ARRAY[1..MAX_MOVER] OF ST_MOVE_DATA;
  _stGearData       : REFERENCE TO ARRAY[1..MAX_MOVER] OF ST_GEAR_DATA;

  _eCmd,
  _eCmdOld          : E_MOVER_CTRL;

  _eState           : E_MOVER_STATE;

  _eResult          : E_PROGRESS;
END_VAR

IF NOT Check() THEN RETURN; END_IF

_stMsg.eDevice                := e_Device.Mover + _nMoverId;

// copy to local for debug
_eCmd                         := _stCtrl[_nMoverId].Cmd;

// cyclic check for command change
// get state for cmd
IF (_eCmd <> _eCmdOld)
THEN
  // get matching sdtate for Ctrl.Cmd
  _eState                     := Cmd(_eCmd);
  _eCmdOld                    := _eCmd;
END_IF


CASE _eResult
OF
  E_PROGRESS.PROGRESS_INVALID:
    _stState[_nMoverId].State := E_MOVER_STATE.MOVER_NULL;

  E_PROGRESS.PROGRESS_ERROR:
    _stState[_nMoverId].State := _eState + E_PROGRESS.PROGRESS_ERROR;

  E_PROGRESS.PROGRESS_DONE:
    _stInfo.nErrorId          := 0;
    _stInfo.bMoverError       := FALSE;
    _stState[_nMoverId].State := _eState + E_PROGRESS.PROGRESS_DONE;

ELSE
  // work in progress
  // update progress for extern use
  _stState[_nMoverId].State   := _eState + _eResult;

  CASE _eState
  OF
    E_MOVER_STATE.MOVER_ENABLE:
      _eResult                := Enable(TRUE);
  
    E_MOVER_STATE.MOVER_DISABLE:
      _eResult                := Disable(TRUE);
  
    E_MOVER_STATE.MOVER_MOVE_TO_POS:
      _eResult                := MoveToPos(TRUE, _stMoveData[_nMoverId]);
  
    E_MOVER_STATE.MOVER_MOVE_TO_POS_CA:
      _eResult                := MoveToPosCa(TRUE, _stMoveData[_nMoverId]);
  
    E_MOVER_STATE.MOVER_SEND_TO_POS_CA:
      _eResult                := SendToModuloPosCa(TRUE, _stMoveData[_nMoverId]);
  
    E_MOVER_STATE.MOVER_HALT:
      _eResult                := Halt(TRUE, _stMoveData[_nMoverId]);
  
    E_MOVER_STATE.MOVER_GEAR_IN:
      _eResult                := GearIn(TRUE, _stMoveData[_nMoverId], _stGearData[_nMoverId]);
  
    E_MOVER_STATE.MOVER_GEAR_IN_POS_CA:
      _eResult                := GearInPosCa(TRUE, _stMoveData[_nMoverId], _stGearData[_nMoverId]);
  
    E_MOVER_STATE.MOVER_GEAR_OUT:
      _eResult                := GearOut(TRUE);
  
    E_MOVER_STATE.MOVER_RESET:
      _eResult                := Reset(TRUE);
  ELSE
      _eResult                := E_PROGRESS.PROGRESS_INVALID;
  END_CASE
END_CASE

METHOD PRIVATE Check : BOOL

// The thing that should not be

IF NOT (_nMoverId > 0)
THEN
  _sState                     := 'Mover: missing ID';
  RETURN;
END_IF

IF NOT __ISVALIDREF(_stCtrl)
THEN
  _sState                     := 'Ctrl: missing pointer';
  RETURN;
END_IF

IF NOT __ISVALIDREF(_stState)
THEN
  _sState                     := 'State: missing pointer';
  RETURN;
END_IF

IF NOT __ISVALIDREF(_Mover)
THEN
  _sState                     := 'Mover: missing pointer';
  RETURN;
END_IF

IF NOT __ISVALIDREF(_rLastPosition)
THEN
  _sState                     := '_rLastPosition: missing pointer';
  RETURN;
END_IF

IF NOT __ISVALIDREF(_rLastGap)
THEN
  _sState                     := '_rLastGap: missing pointer';
  RETURN;
END_IF

IF NOT __ISVALIDREF(_stInfo)
THEN
  _sState                     := '_stInfo: missing pointer';
  RETURN;
END_IF

IF NOT __ISVALIDREF(_stGearData)
THEN
  _sState                     := '_stGearData: missing pointer';
  RETURN;
END_IF

IF NOT __ISVALIDREF(_stMoveData)
THEN
  _sState                     := '_stMoveData: missing pointer';
  RETURN;
END_IF

_sState                       := 'CHECK_DONE';
Check                         := TRUE;
END_METHOD

METHOD PRIVATE Cmd : E_MOVER_STATE
VAR_INPUT
  Ctrl      : E_MOVER_CTRL;
END_VAR
VAR_INST
  _eState   : E_MOVER_STATE;
END_VAR
IF NOT Check() THEN Cmd := E_MOVER_STATE.MOVER_NULL;  RETURN; END_IF


CASE Ctrl
OF
  E_MOVER_CTRL.MOVER_ENABLE:
    _eResult          := Enable(FALSE);
    _eState           := E_MOVER_STATE.MOVER_ENABLE;

  E_MOVER_CTRL.MOVER_DISABLE:
    _eResult          := Disable(FALSE);
    _eState           := E_MOVER_STATE.MOVER_DISABLE;

  E_MOVER_CTRL.MOVER_MOVE_TO_POS:
    _eResult          := MoveToPos(FALSE, _stMoveData[_nMoverId]);
    _eState           := E_MOVER_STATE.MOVER_MOVE_TO_POS;

  E_MOVER_CTRL.MOVER_MOVE_TO_POS_CA:
    _eResult          := MoveToPosCa(FALSE, _stMoveData[_nMoverId]);
    _eState           := E_MOVER_STATE.MOVER_MOVE_TO_POS_CA;

  E_MOVER_CTRL.MOVER_SEND_TO_POS_CA:
    _eResult          := SendToModuloPosCa(FALSE, _stMoveData[_nMoverId]);
    _eState           := E_MOVER_STATE.MOVER_SEND_TO_POS_CA;

  E_MOVER_CTRL.MOVER_HALT:
    _eResult          := Halt(FALSE, _stMoveData[_nMoverId]);
    _eState           := E_MOVER_STATE.MOVER_HALT;

  E_MOVER_CTRL.MOVER_GEAR_IN:
    _eResult          := GearIn(FALSE,  _stMoveData[_nMoverId], _stGearData[_nMoverId]);
    _eState           := E_MOVER_STATE.MOVER_GEAR_IN;

  E_MOVER_CTRL.MOVER_GEAR_IN_POS_CA:
    _eResult          := GearInPosCa(FALSE, _stMoveData[_nMoverId], _stGearData[_nMoverId]);
    _eState           := E_MOVER_STATE.MOVER_GEAR_IN_POS_CA;

  E_MOVER_CTRL.MOVER_GEAR_OUT:
    _eResult          := GearOut(FALSE);
    _eState           := E_MOVER_STATE.MOVER_GEAR_OUT;

  E_MOVER_CTRL.MOVER_RESET:
    _eResult          := Reset(FALSE);
    _eState           := E_MOVER_STATE.MOVER_RESET;

ELSE
    _eResult          := E_PROGRESS.PROGRESS_INVALID; 
    _eState           := E_MOVER_STATE.MOVER_NULL;
END_CASE

Cmd                   := _eState;
END_METHOD

PROPERTY Ctrl : REFERENCE TO ARRAY[1..MAX_MOVER] OF ST_MOVER_CTRL
SET
_stCtrl ref= Ctrl;
END_SET
END_PROPERTY

PROPERTY GearData : reference TO ARRAY[1..MAX_MOVER] OF ST_GEAR_DATA
SET
_stGearData REF= GearData;
END_SET
END_PROPERTY

PROPERTY MoveData : reference TO ARRAY[1..MAX_MOVER] OF st_move_data
SET
_stMoveData REF= MoveData;
END_SET
END_PROPERTY

PROPERTY State : REFERENCE TO ARRAY[1..MAX_MOVER] OF ST_MOVER_STATE
SET
_stState ref= State;
END_SET
END_PROPERTY

END_FUNCTION_BLOCK

// ---- XTS/Mover/fb_Mover.TcPOU
//---------------------------------------------------------------------------------------------------------------
//
//  HAUD 2023.12.19
//
//  - XTS_TRANSPORT_LAYER
//
//  fb_Mover
//  - all positioning input is modulo value
//  - wrap MC function blocks
//
//
//---------------------------------------------------------------------------------------------------------------
// This SOFTWARE is provided as an Example by THE PROVIDER "as is" and "with all faults." THE PROVIDER makes no 
// representations or warranties of any kind concerning the safety, suitability, lack of viruses, inaccuracies, 
// typographical errors, or other harmful components of this SOFTWARE. There are inherent dangers in the use of 
// any software, and you are solely responsible for determining whether this SOFTWARE is compatible with your 
// equipment and other software installed on your equipment. You are also solely responsible for the protection 
// of your equipment and backup of your data, and THE PROVIDER will not be liable for any damages you may suffer 
// in connection with using, modifying, or distributing this SOFTWARE.
//---------------------------------------------------------------------------------------------------------------
FUNCTION_BLOCK fb_Mover IMPLEMENTS I_XtsTransport_Mover
VAR
  _nMoverId         : UINT;

  _sState           : STRING;

  _Master,
  _Mover            : REFERENCE TO AXIS_REF;
  _rLastPosition    : REFERENCE TO LREAL;
  _rLastGap         : REFERENCE TO LREAL;

  _RailLength       : LREAL;
  _nSyncStrategy    : Tc3_Mc3Definitions.MC_SYNC_STRATEGY := Tc3_Mc3Definitions.MC_SYNC_STRATEGY.mcSyncStrategySlow; // minimal movement with this strategy 

  // mover compact axis information
  _stInfo           : REFERENCE TO ST_MOVER_INFO; // ActPos, Enable, ...

  _bError           : BOOL;   // used in Cycle()
  _nErrorIdMover,             // used in Cycle()
  _nErrorIdPower    : UDINT;  // used in Cycle()

  //---------------------------------------------------------------------------
  // MC2 and CA function blocks
  //---------------------------------------------------------------------------
  _wMoverState      : DWORD;

  _fbMoveAbsCa      : Tc3_McCollisionAvoidance.MC_MoveAbsoluteCA;
  _fbGearInPosCa    : Tc3_McCollisionAvoidance.MC_GearInPosCA;
  _fbHaltCa         : Tc3_McCollisionAvoidance.MC_HaltCA;

  _fbMoveAbs        : Tc2_MC2.MC_MoveAbsolute;
  _fbHalt           : Tc2_MC2.MC_Halt;
  _fbReset          : Tc2_MC2.MC_Reset;
  _fbStop           : Tc2_MC2.MC_Stop;

  _fbGearIn         : Tc2_MC2.MC_GearIn;
  _fbGearOut        : Tc2_MC2.MC_GearOut;

  _fbPower          : Tc2_MC2.MC_Power;

  _stMsg            : ST_Message;
  _eMessageLevel    : E_MessageType;
END_VAR

METHOD Check : BOOL
// check The thing that should not be

IF NOT (_nMoverId > 0)
THEN
  _sState                     := 'Mover: missing ID';
  RETURN;
END_IF

IF NOT __ISVALIDREF(_Mover)
THEN
  _sState                     := 'Mover: missing pointer';
  RETURN;
END_IF

IF NOT __ISVALIDREF(_rLastPosition)
THEN
  _sState                     := '_rLastPosition: missing pointer';
  RETURN;
END_IF

IF NOT __ISVALIDREF(_rLastGap)
THEN
  _sState                     := '_rLastGap: missing pointer';
  RETURN;
END_IF

IF NOT __ISVALIDREF(_stInfo)
THEN
  _sState                     := '_stInfo: missing pointer';
  RETURN;
END_IF

_sState                       := 'CHECK_DONE';
Check                         := TRUE;
END_METHOD

METHOD Cycle : E_PROGRESS
VAR_INST
  _eState             : E_PROGRESS;

  _rtrigMoverError,
  _rtrigPowerError    : Tc2_Standard.R_TRIG;
END_VAR
IF NOT Check() THEN Cycle := E_PROGRESS.PROGRESS_ERROR; RETURN; END_IF

_stMsg.eDevice            := e_Device.Mover + _nMoverId;

//-----------------------------------------------------------------------------------------------
// cyclic NC mapping
//-----------------------------------------------------------------------------------------------
_Mover();
//-----------------------------------------------------------------------------------------------


//-----------------------------------------------------------------------------------------------
// cyclic MC_Power
//-----------------------------------------------------------------------------------------------
_fbPower(
        Axis              := _Mover, 
        Enable_Positive   := TRUE, 
        Enable_Negative   := TRUE, 
        BufferMode        := MC_BufferMode.MC_Aborting);

_rtrigPowerError(CLK := _fbPower.Error);
_rtrigMoverError(CLK := _Mover.Status.Error); 

IF _rtrigMoverError.Q
THEN
  _bError                 := TRUE;  // deleted by Reset()
  // catch error
  _nErrorIdMover          := _Mover.Status.ErrorID;
  _stInfo.nErrorId        := _nErrorIdMover;

  _stMsg.eType            := E_MessageType.eMessageError;
  _stMsg.eSubdevice       := e_Subdevice.AxisControl;
  _stMsg.iErrorNumber     := _nErrorIdMover;
  _stMsg.sText            := 'Axis Error';
  f_MessageSet(_stMsg);
END_IF

IF _rtrigPowerError.Q
THEN
  _bError                 := TRUE;  // deleted by Reset()
  // catch error
  _nErrorIdPower          := _fbPower.ErrorID;
  _stInfo.nErrorId        := _nErrorIdPower;

  _stMsg.eType            := E_MessageType.eMessageError;
  _stMsg.eSubdevice       := e_Subdevice.AxisControl;
  _stMsg.iErrorNumber     := _nErrorIdMover;
  _stMsg.sText            := 'Axis Error';
  f_MessageSet(_stMsg);
END_IF
//-----------------------------------------------------------------------------------------------

//-----------------------------------------------------------------------------------------------
// cyclic state
//-----------------------------------------------------------------------------------------------
IF NOT _Mover.Status.ControlLoopClosed
THEN
  _eState                       := E_PROGRESS.PROGRESS_INIT;
ELSE
  _eState                       := E_PROGRESS.PROGRESS_WORKING;
END_IF
 
IF _bError
THEN
  _eState                       := E_PROGRESS.PROGRESS_ERROR;
END_IF
//-----------------------------------------------------------------------------------------------


//-----------------------------------------------------------------------------
// cyclic Mover info data
// get collision avoiding information from cyclic interface
//-----------------------------------------------------------------------------------------------
memcpy(ADR(_wMoverState), ADR(_Mover.NcToPlc.StateDWord2), SIZEOF(_wMoverState));

_stInfo.bMoverEnabled           := _Mover.Status.ControlLoopClosed;
_stInfo.bMoverError             := _bError;
_stInfo.bMoverCoupled           := _Mover.Status.Coupled;
_stInfo.bMoverStandstill        := _Mover.Status.NotMoving;
_stInfo.bMoverAvoidingCollision := _wMoverState.0;

_stInfo.rModuloActPos           := TO_REAL(_Mover.NcToPlc.ModuloActPos);
_stInfo.rAbsActPos              := TO_REAL(_Mover.NcToPlc.ActPos);

_stInfo.rModuloTargetPos        := TO_REAL(Tc2_Math.LMOD(_rLastPosition, _RailLength));
_stInfo.rAbsTargetPos           := TO_REAL(_rLastPosition);

IF (_Mover.NcToPlc.ActPos < _rLastPosition + 0.05) AND
   (_Mover.NcToPlc.ActPos > _rLastPosition - 0.05)
THEN
  _stInfo.bMoverInTarget        := TRUE;
ELSE
  _stInfo.bMoverInTarget        := FALSE;
END_IF
//-----------------------------------------------------------------------------

Cycle                           := _eState;
END_METHOD

METHOD Disable : E_PROGRESS
VAR_INPUT
  Execute             : BOOL;
END_VAR
VAR_INST
  _nErrorId           : UDINT;
  _eState             : E_PROGRESS;
END_VAR
IF NOT Execute THEN _eState  := E_PROGRESS.PROGRESS_INIT; END_IF 
IF NOT Check() THEN Disable  := E_PROGRESS.PROGRESS_ERROR; RETURN; END_IF


CASE _eState
OF
  E_PROGRESS.PROGRESS_INIT:
    IF Execute
    THEN
      _nErrorId               := 0;
      _eState                 := E_PROGRESS.PROGRESS_BUSY;
    END_IF
END_CASE
//-----------------------------------------------------------------------------
//-----------------------------------------------------------------------------
CASE _eState
OF
  E_PROGRESS.PROGRESS_BUSY:
    _eState                   := E_PROGRESS.PROGRESS_PREPARE;
    _fbPower.Enable           := FALSE;
END_CASE
//-----------------------------------------------------------------------------
//-----------------------------------------------------------------------------
CASE _eState
OF
  E_PROGRESS.PROGRESS_PREPARE:
    IF (_fbPower.Error)
    THEN
      _eState                 := E_PROGRESS.PROGRESS_ERROR;
      _nErrorId               := _fbPower.ErrorId;

      _stMsg.eType            := E_MessageType.eMessageError;
      _stMsg.eSubdevice       := e_Subdevice.fbPower;
      _stMsg.iErrorNumber     := _nErrorId;
      _stMsg.sText            := concat('Axis Disable: ', TO_STRING(_eState));
      f_MessageSet(_stMsg);

    ELSIF NOT (_Mover.Status.ControlLoopClosed)
    THEN
      _eState                 := E_PROGRESS.PROGRESS_DONE;

      IF (_eMessageLevel > E_MessageType.eMessageError)
      THEN
        _stMsg.eType          := E_MessageType.eMessageInfo;
        _stMsg.eSubdevice     := e_Subdevice.fbPower;
        _stMsg.iErrorNumber   := 0;
        _stMsg.sText          := concat('Axis Disable: ', TO_STRING(_eState));
        f_MessageSet(_stMsg);
      END_IF
    END_IF
END_CASE
//-----------------------------------------------------------------------------
//-----------------------------------------------------------------------------

Disable                       := _eState;
END_METHOD

METHOD Enable : E_PROGRESS
VAR_INPUT
  Execute             : BOOL;
END_VAR
VAR_INST
  _nErrorId           : UDINT;
  _eState             : E_PROGRESS;
END_VAR
IF NOT Execute THEN _eState  := E_PROGRESS.PROGRESS_INIT; END_IF 
IF NOT Check() THEN Enable   := E_PROGRESS.PROGRESS_ERROR; RETURN; END_IF


CASE _eState
OF
  E_PROGRESS.PROGRESS_INIT:
    IF Execute
    THEN
      _nErrorId               := 0;
      _eState                 := E_PROGRESS.PROGRESS_BUSY;
    END_IF
END_CASE
//-----------------------------------------------------------------------------
//-----------------------------------------------------------------------------
CASE _eState
OF
  E_PROGRESS.PROGRESS_BUSY:
    _eState                   := E_PROGRESS.PROGRESS_PREPARE;
    _fbPower.Enable           := TRUE;
END_CASE
//-----------------------------------------------------------------------------
//-----------------------------------------------------------------------------
CASE _eState
OF
  E_PROGRESS.PROGRESS_PREPARE:
    IF (_fbPower.Error)
    THEN
      _eState                 := E_PROGRESS.PROGRESS_ERROR;
      _nErrorId               := _fbPower.ErrorId;
      _stInfo.nErrorId        := _nErrorId;

      _stMsg.eType            := E_MessageType.eMessageError;
      _stMsg.eSubdevice       := e_Subdevice.fbPower;
      _stMsg.iErrorNumber     := _nErrorId;
      _stMsg.sText            := concat('Axis Enable: ', TO_STRING(_eState));
      f_MessageSet(_stMsg);

    ELSIF (_Mover.Status.ControlLoopClosed)
    THEN
      _eState                 := E_PROGRESS.PROGRESS_DONE;

      IF (_eMessageLevel > E_MessageType.eMessageError)
      THEN
        _stMsg.eType          := E_MessageType.eMessageInfo;
        _stMsg.eSubdevice     := e_Subdevice.fbPower;
        _stMsg.iErrorNumber   := _nErrorId;
        _stMsg.sText          := concat('Axis Enable: ', TO_STRING(_eState));
        f_MessageSet(_stMsg);
      END_IF
    END_IF
END_CASE
//-----------------------------------------------------------------------------
//-----------------------------------------------------------------------------

Enable                   := _eState;
END_METHOD

METHOD GearIn : E_PROGRESS;
VAR_INPUT
  Execute             : BOOL;
  stMoveData          : ST_MOVE_DATA;
  stGearData          : ST_GEAR_DATA;
END_VAR
VAR_INST
  _nErrorId           : UDINT;
  _eState             : E_PROGRESS;
END_VAR
IF NOT Execute THEN _eState  := E_PROGRESS.PROGRESS_INIT; END_IF 
IF NOT Check() THEN GearIn   := E_PROGRESS.PROGRESS_ERROR; RETURN; END_IF


CASE _eState
OF
  E_PROGRESS.PROGRESS_INIT:
    IF Execute
    THEN
      _nErrorId               := 0;
      _eState                 := E_PROGRESS.PROGRESS_BUSY;

      IF NOT __ISVALIDREF(_Master)
      THEN
        _bError               := TRUE;
        _nErrorId             := 666;
        _eState               := E_PROGRESS.PROGRESS_ERROR;

        _stMsg.eType          := E_MessageType.eMessageError;
        _stMsg.eSubdevice     := e_Subdevice.fbGearIn;
        _stMsg.iErrorNumber   := _nErrorId;
        _stMsg.sText          := concat('Invalid Master Ref: ', TO_STRING(_eState));
        f_MessageSet(_stMsg);
      END_IF
    END_IF
END_CASE
//-----------------------------------------------------------------------------
//-----------------------------------------------------------------------------
CASE _eState
OF
  E_PROGRESS.PROGRESS_BUSY:
    _eState                   := E_PROGRESS.PROGRESS_PREPARE;
    _fbPower.Override         := stMoveData.rOverride;

    _fbGearIn(
            Master            := _Master, 
            Slave             := _Mover,
            Execute           := FALSE,
            RatioNumerator    := stGearData.rGearNumerator,
            RatioDenominator  := stGearData.iGearDenumerator, 
            Acceleration      := stMoveData.rAcc, 
            Deceleration      := stMoveData.rAcc, 
            Jerk              := stMoveData.rJerk, 
            BufferMode        := Tc2_MC2.MC_BufferMode.MC_Aborting);
END_CASE
//-----------------------------------------------------------------------------
//-----------------------------------------------------------------------------
CASE _eState
OF
  E_PROGRESS.PROGRESS_PREPARE:
    _fbGearIn(
            Master            := _Master, 
            Slave             := _Mover,
            Execute           := TRUE);

    IF _fbGearIn.Error
    THEN
      _bError                 := TRUE;
      _nErrorId               := _fbGearIn.ErrorID;
      _eState                 := E_PROGRESS.PROGRESS_ERROR;

      _stMsg.eType            := E_MessageType.eMessageError;
      _stMsg.eSubdevice       := e_Subdevice.fbGearIn;
      _stMsg.iErrorNumber     := _nErrorId;
      _stMsg.sText            := TO_STRING(_eState);
      f_MessageSet(_stMsg);

    ELSIF _fbGearIn.InGear
    THEN
      _eState                 := E_PROGRESS.PROGRESS_DONE;

      IF (_eMessageLevel > E_MessageType.eMessageError)
      THEN
        _stMsg.eType          := E_MessageType.eMessageInfo;
        _stMsg.eSubdevice     := e_Subdevice.fbGearIn;
        _stMsg.iErrorNumber   := _nErrorId;
        _stMsg.sText          := TO_STRING(_eState);
        f_MessageSet(_stMsg);
      END_IF
    END_IF
END_CASE
//-----------------------------------------------------------------------------
//-----------------------------------------------------------------------------
CASE _eState
OF
  E_PROGRESS.PROGRESS_ERROR,
  E_PROGRESS.PROGRESS_DONE:
    _stInfo.nErrorId          := _nErrorId;
    _fbGearIn(
            Master            := _Master, 
            Slave             := _Mover,
            Execute           := FALSE);
END_CASE
//-----------------------------------------------------------------------------
//-----------------------------------------------------------------------------

GearIn                        := _eState;
END_METHOD

METHOD GearInPosCa : E_PROGRESS
VAR_INPUT
  Execute             : BOOL;
  stMoveData          : ST_MOVE_DATA;
  stGearData          : ST_GEAR_DATA;  
END_VAR
VAR_INST
  _nErrorId           : UDINT;
  _rPosLate,
  _rPos               : LREAL;
  _eState             : E_PROGRESS;
END_VAR
IF NOT Execute THEN _eState       := E_PROGRESS.PROGRESS_INIT; END_IF 
IF NOT Check() THEN GearInPosCa   := E_PROGRESS.PROGRESS_ERROR; RETURN; END_IF


CASE _eState
OF
  E_PROGRESS.PROGRESS_INIT:
    IF Execute
    THEN
      _rPosLate               := 0.0;
      _nErrorId               := 0;
      _eState                 := E_PROGRESS.PROGRESS_BUSY;

      IF NOT __ISVALIDREF(_Master)
      THEN
        _bError               := TRUE;
        _nErrorId             := 666;
        _eState               := E_PROGRESS.PROGRESS_ERROR;

        _stMsg.eType          := E_MessageType.eMessageError;
        _stMsg.eSubdevice     := e_Subdevice.fbGearInPosCa;
        _stMsg.iErrorNumber   := _nErrorId;
        _stMsg.sText          := concat('Invalid Master Ref: ', TO_STRING(_eState));
        f_MessageSet(_stMsg);

      ELSIF (_Mover.NcToPlc.ModuloActPos > stGearData.rModuloSyncPosSlave + stMoveData.rDelta)
      THEN
        _bError               := TRUE;
        _rPosLate             := _Mover.NcToPlc.ModuloActPos;
        _rPos                 := stGearData.rModuloSyncPosSlave + stMoveData.rDelta;

        _nErrorId             := 667;
        _eState               := E_PROGRESS.PROGRESS_ERROR;

        _stMsg.eType          := E_MessageType.eMessageError;
        _stMsg.eSubdevice     := e_Subdevice.fbGearInPosCa;
        _stMsg.iErrorNumber   := _nErrorId;
        _stMsg.sText          := concat('ModuloActPosMover: ', TO_STRING(_rPosLate));
        _stMsg.sText          := concat(_stMsg.sText, '; ModuloSyncPosSlave + stMoveData.Delta: ');
        _stMsg.sText          := concat(_stMsg.sText, TO_STRING(_rPos));
        f_MessageSet(_stMsg);
      END_IF
    END_IF
END_CASE
//-----------------------------------------------------------------------------
//-----------------------------------------------------------------------------
CASE _eState
OF
  E_PROGRESS.PROGRESS_BUSY:
    _eState                   := E_PROGRESS.PROGRESS_PREPARE;

    _fbPower.Override         := stMoveData.rOverride;

    _fbGearInPosCa(
        Master                := _Master, 
        Slave                 := _Mover, 
        Execute               := FALSE, 
        ContinuousUpdate      := TRUE, 
        RatioNumerator        := stGearData.rGearNumerator, 
        RatioDenumerator      := stGearData.iGearDenumerator, 

        MasterSyncPosition    := _Master.NcToPlc.ActPos 
                               + stGearData.rDeltaToMasterPos,                            // absolute position

        SlaveSyncPosition     := ABS(_Mover.NcToPlc.ModuloActTurns)*_RailLength
                               + stGearData.rModuloSyncPosSlave,                          // absolute position

        SyncStrategy          := _nSyncStrategy,  
        SyncMode              := Tc3_Mc3Definitions.MC_SYNC_MODE.mcSyncModeNonModulo,     // all positions as absolute value
        MasterStartDistance   := stGearData.rMasterStartDistance,                         // if <> 0 --> master has to move before this fb does anything
        Velocity              := stMoveData.rVelo, 
        Acceleration          := stMoveData.rAcc, 
        Deceleration          := stMoveData.rAcc, 
        Jerk                  := stMoveData.rJerk, 
        Gap                   := stMoveData.rGap, 
        BufferMode            := Tc3_Mc3Definitions.MC_BUFFER_MODE.mcAborting);

        IF (_eMessageLevel > E_MessageType.eMessageInfo)
        THEN
          _stMsg.eType        := E_MessageType.eMessageVerbose;
          _stMsg.eSubdevice   := e_Subdevice.fbGearInPosCa;
          _stMsg.iErrorNumber := _nErrorId;
          _stMsg.sText        := TO_STRING(_eState);
          f_MessageSet(_stMsg);
        END_IF
END_CASE
//-----------------------------------------------------------------------------
//-----------------------------------------------------------------------------
CASE _eState
OF
  E_PROGRESS.PROGRESS_PREPARE:
    _fbGearInPosCa(
        Master                := _Master, 
        Slave                 := _Mover, 
        Execute               := TRUE, 
        ContinuousUpdate      := TRUE);

    IF _fbGearInPosCa.Error
    THEN
      _bError                 := TRUE;
      _nErrorId               := _fbGearInPosCa.ErrorId;
      _stInfo.nErrorId        := _nErrorId;
      _fbGearInPosCa(
        Master                := _Master, 
        Slave                 := _Mover, 
        Execute               := FALSE, 
        ContinuousUpdate      := TRUE);

      _eState                 := E_PROGRESS.PROGRESS_ERROR;

      _stMsg.eType          := E_MessageType.eMessageError;
      _stMsg.eSubdevice     := e_Subdevice.fbGearInPosCa;
      _stMsg.iErrorNumber   := _nErrorId;
      _stMsg.sText          := TO_STRING(_eState);
      f_MessageSet(_stMsg);

    ELSIF _fbGearInPosCa.CommandAborted
    THEN
      _bError                 := TRUE;
      _eState                 := E_PROGRESS.PROGRESS_OCCUPIED;

      _stMsg.eType            := E_MessageType.eMessageWarning;
      _stMsg.eSubdevice       := e_Subdevice.fbGearInPosCa;
      _stMsg.iErrorNumber     := _nErrorId;
      _stMsg.sText            := TO_STRING(_eState);
      f_MessageSet(_stMsg);

    ELSIF _fbGearInPosCa.InSync
    THEN
      _eState                 := E_PROGRESS.PROGRESS_DONE;

      IF (_eMessageLevel > E_MessageType.eMessageError)
      THEN
        _stMsg.eType          := E_MessageType.eMessageInfo;
        _stMsg.eSubdevice     := e_Subdevice.fbGearInPosCa;
        _stMsg.iErrorNumber   := _nErrorId;
        _stMsg.sText          := TO_STRING(_eState);
        f_MessageSet(_stMsg);
      END_IF
      _fbGearInPosCa(
        Master                := _Master, 
        Slave                 := _Mover, 
        Execute               := FALSE, 
        ContinuousUpdate      := TRUE);
    END_IF
END_CASE
//-----------------------------------------------------------------------------
//-----------------------------------------------------------------------------

GearInPosCa                   := _eState;
END_METHOD

METHOD GearOut : E_PROGRESS
VAR_INPUT
  Execute             : BOOL;
END_VAR
VAR_INST
  _nErrorId           : UDINT;
  _eState             : E_PROGRESS;
END_VAR
IF NOT Execute THEN _eState  := E_PROGRESS.PROGRESS_INIT; END_IF 
IF NOT Check() THEN GearOut  := E_PROGRESS.PROGRESS_ERROR; RETURN; END_IF


CASE _eState
OF
  E_PROGRESS.PROGRESS_INIT:
    IF Execute
    THEN
      _nErrorId               := 0;
      _eState                 := E_PROGRESS.PROGRESS_BUSY;
    END_IF
END_CASE
//-----------------------------------------------------------------------------
//-----------------------------------------------------------------------------
CASE _eState
OF
  E_PROGRESS.PROGRESS_BUSY:
    _eState                   := E_PROGRESS.PROGRESS_PREPARE;
    _fbGearOut(
            Slave             := _Mover, 
            Execute           := FALSE);

    IF (_eMessageLevel > E_MessageType.eMessageError)
    THEN
      _stMsg.eType            := E_MessageType.eMessageInfo;
      _stMsg.eSubdevice       := e_Subdevice.fbGearOut;
      _stMsg.iErrorNumber     := _nErrorId;
      _stMsg.sText            := TO_STRING(_eState);
      f_MessageSet(_stMsg);
    END_IF
END_CASE
//-----------------------------------------------------------------------------
//-----------------------------------------------------------------------------
CASE _eState
OF
  E_PROGRESS.PROGRESS_PREPARE:
    _fbGearOut(
            Slave             := _Mover, 
            Execute           := TRUE);

    IF _fbGearOut.Error
    THEN
      _bError                 := TRUE;
      _nErrorId               := _fbGearOut.ErrorID;
      _eState                 := E_PROGRESS.PROGRESS_ERROR;

      _stMsg.eType            := E_MessageType.eMessageError;
      _stMsg.eSubdevice       := e_Subdevice.fbGearOut;
      _stMsg.iErrorNumber     := _nErrorId;
      _stMsg.sText            := TO_STRING(_eState);
      f_MessageSet(_stMsg);

    ELSIF (_Mover.NcToPlc.CoupleState = 0)
    THEN
      _eState                 := E_PROGRESS.PROGRESS_DONE;

      IF (_eMessageLevel > E_MessageType.eMessageError)
      THEN
        _stMsg.eType          := E_MessageType.eMessageInfo;
        _stMsg.eSubdevice     := e_Subdevice.fbGearOut;
        _stMsg.iErrorNumber   := _nErrorId;
        _stMsg.sText          := TO_STRING(_eState);
        f_MessageSet(_stMsg);
      END_IF
    END_IF
END_CASE
//-----------------------------------------------------------------------------
//-----------------------------------------------------------------------------
CASE _eState
OF
  E_PROGRESS.PROGRESS_ERROR,
  E_PROGRESS.PROGRESS_DONE:
    _stInfo.nErrorId          := _nErrorId;
    _fbGearOut(
            Slave             := _Mover, 
            Execute           := FALSE);
END_CASE
//-----------------------------------------------------------------------------
//-----------------------------------------------------------------------------

GearOut                       := _eState;
END_METHOD

METHOD Halt : E_PROGRESS
VAR_INPUT
  Execute             : BOOL;
  stMoveData          : ST_MOVE_DATA;
END_VAR
VAR_INST
  _nErrorId           : UDINT;
  _eState             : E_PROGRESS;
END_VAR
IF NOT Execute 
THEN 
	_eState := E_PROGRESS.PROGRESS_INIT; 
END_IF 
IF NOT Check() 
THEN 
	Halt := E_PROGRESS.PROGRESS_ERROR; 
	RETURN; 
END_IF


CASE _eState
OF
  E_PROGRESS.PROGRESS_INIT:
    IF Execute
    THEN
      _nErrorId               := 0;
      _eState                 := E_PROGRESS.PROGRESS_BUSY;
    END_IF
END_CASE
//-----------------------------------------------------------------------------
//-----------------------------------------------------------------------------
CASE _eState
OF
  E_PROGRESS.PROGRESS_BUSY:
    _eState                   := E_PROGRESS.PROGRESS_PREPARE;
    _fbHalt(
            Axis              := _Mover, 
            Execute           := FALSE, 
            Deceleration      := stMoveData.rAcc, 
            Jerk              := stMoveData.rJerk, 
            BufferMode        := Tc2_MC2.MC_BufferMode.MC_Aborting);

    IF (_eMessageLevel > E_MessageType.eMessageInfo)
    THEN
      _stMsg.eType            := E_MessageType.eMessageVerbose;
      _stMsg.eSubdevice       := e_Subdevice.fbHalt;
      _stMsg.iErrorNumber     := _nErrorId;
      _stMsg.sText            := TO_STRING(_eState);
      f_MessageSet(_stMsg);
    END_IF
END_CASE
//-----------------------------------------------------------------------------
//-----------------------------------------------------------------------------
CASE _eState
OF
  E_PROGRESS.PROGRESS_PREPARE:
    _fbHalt(Axis              := _Mover, 
            Execute           := TRUE, 
            Deceleration      := stMoveData.rAcc, 
            Jerk              := stMoveData.rJerk, 
            BufferMode        := Tc2_MC2.MC_BufferMode.MC_Aborting);

    IF _fbHalt.Error
    THEN
      _bError                 := TRUE;
      _nErrorId               := _fbHalt.ErrorID;
      _eState                 := E_PROGRESS.PROGRESS_ERROR;

      _stMsg.eType            := E_MessageType.eMessageError;
      _stMsg.eSubdevice       := e_Subdevice.fbHalt;
      _stMsg.iErrorNumber     := _nErrorId;
      _stMsg.sText            := TO_STRING(_eState);
      f_MessageSet(_stMsg);

    ELSIF NOT _Mover.Status.Moving
    THEN
      _eState                 := E_PROGRESS.PROGRESS_DONE;

      IF (_eMessageLevel > E_MessageType.eMessageError)
      THEN
        _stMsg.eType          := E_MessageType.eMessageInfo;
        _stMsg.eSubdevice     := e_Subdevice.fbHalt;
        _stMsg.iErrorNumber   := _nErrorId;
        _stMsg.sText          := TO_STRING(_eState);
        f_MessageSet(_stMsg);
      END_IF
    END_IF
END_CASE
//-----------------------------------------------------------------------------
//-----------------------------------------------------------------------------
CASE _eState
OF
  E_PROGRESS.PROGRESS_ERROR,
  E_PROGRESS.PROGRESS_DONE:
    _stInfo.nErrorId          := _nErrorId;
    _fbHalt(
            Axis              := _Mover, 
            Execute           := FALSE);
END_CASE
//-----------------------------------------------------------------------------
//-----------------------------------------------------------------------------

Halt                          := _eState;
END_METHOD

METHOD HaltCa : E_PROGRESS
VAR_INPUT
  Execute             : BOOL;
  stMoveData          : ST_MOVE_DATA;
END_VAR
VAR_INST
  _nErrorId           : UDINT;
  _eState             : E_PROGRESS;
END_VAR
IF NOT Execute 
THEN 
	_eState := E_PROGRESS.PROGRESS_INIT; 
END_IF 
IF NOT Check() 
THEN 
	HaltCa := E_PROGRESS.PROGRESS_ERROR; 
	RETURN; 
END_IF


CASE _eState
OF
  E_PROGRESS.PROGRESS_INIT:
    IF Execute
    THEN
      _nErrorId               := 0;
      _eState                 := E_PROGRESS.PROGRESS_BUSY;
    END_IF
END_CASE
//-----------------------------------------------------------------------------
//-----------------------------------------------------------------------------
CASE _eState
OF
  E_PROGRESS.PROGRESS_BUSY:
    _eState                   := E_PROGRESS.PROGRESS_PREPARE;
    _fbHaltCa(
            Axis              := _Mover, 
            Execute           := FALSE, 
            Deceleration      := stMoveData.rAcc, 
            Jerk              := stMoveData.rJerk, 
            Gap               := stMoveData.rGap);

    IF (_eMessageLevel > E_MessageType.eMessageInfo)
    THEN
      _stMsg.eType            := E_MessageType.eMessageVerbose;
      _stMsg.eSubdevice       := e_Subdevice.fbHaltCa;
      _stMsg.iErrorNumber     := _nErrorId;
      _stMsg.sText            := TO_STRING(_eState);
      f_MessageSet(_stMsg);
    END_IF
END_CASE
//-----------------------------------------------------------------------------
//-----------------------------------------------------------------------------
CASE _eState
OF
  E_PROGRESS.PROGRESS_PREPARE:
    _fbHaltCa(
            Axis              := _Mover, 
            Execute           := TRUE, 
            Deceleration      := stMoveData.rAcc, 
            Jerk              := stMoveData.rJerk, 
            Gap               := stMoveData.rGap);

    IF _fbHaltCa.Error
    THEN
      _bError                 := TRUE;
      _nErrorId               := _fbHalt.ErrorID;
      _eState                 := E_PROGRESS.PROGRESS_ERROR;

      _stMsg.eType            := E_MessageType.eMessageError;
      _stMsg.eSubdevice       := e_Subdevice.fbHaltCa;
      _stMsg.iErrorNumber     := _nErrorId;
      _stMsg.sText            := TO_STRING(_eState);
      f_MessageSet(_stMsg);

    ELSIF NOT _Mover.Status.Moving
    THEN
      _eState                 := E_PROGRESS.PROGRESS_DONE;

      IF (_eMessageLevel > E_MessageType.eMessageError)
      THEN
        _stMsg.eType          := E_MessageType.eMessageInfo;
        _stMsg.eSubdevice     := e_Subdevice.fbHaltCa;
        _stMsg.iErrorNumber   := _nErrorId;
        _stMsg.sText          := TO_STRING(_eState);
        f_MessageSet(_stMsg);
      END_IF
    END_IF
END_CASE
//-----------------------------------------------------------------------------
//-----------------------------------------------------------------------------
CASE _eState
OF
  E_PROGRESS.PROGRESS_ERROR,
  E_PROGRESS.PROGRESS_DONE:
    _stInfo.nErrorId          := _nErrorId;
    _fbHaltCa(
            Axis              := _Mover, 
            Execute           := FALSE);
END_CASE
//-----------------------------------------------------------------------------
//-----------------------------------------------------------------------------

HaltCa                          := _eState;
END_METHOD

PROPERTY LastGap : REFERENCE to lreal
SET
_rLastGap REF= LastGap;
END_SET
END_PROPERTY

PROPERTY LastPosition : REFERENCE to LREAL
SET
_rLastPosition REF= LastPosition;
END_SET
END_PROPERTY

PROPERTY Master : REFERENCE to AXIS_REF
SET
_Master REF= Master;
END_SET
END_PROPERTY

PROPERTY MessageLevel : e_messagetype
SET
_eMessageLevel := MessageLevel;
END_SET
END_PROPERTY

PROPERTY ModuloTurn : dint
GET
ModuloTurn := _Mover.NcToPlc.ModuloSetTurns;
END_GET
END_PROPERTY

PROPERTY Mover : REFERENCE to AXIS_REF
SET
_Mover REF= Mover;
END_SET
END_PROPERTY

PROPERTY MoverId : uint
SET
_nMoverId := MoverId;
END_SET
END_PROPERTY

PROPERTY MoverInfo : REFERENCE to ST_MOVER_INFO
SET


	_stInfo ref= MoverInfo;
END_SET
END_PROPERTY

METHOD MoveToPos : E_PROGRESS
VAR_INPUT
  Execute             : BOOL;
  stMoveData          : ST_MOVE_DATA;
END_VAR
VAR_INST
  _nErrorId           : UDINT;
  _rDelta,
  _rPos               : LREAL;
  _eState             : E_PROGRESS;
END_VAR
IF NOT Execute THEN _eState  := E_PROGRESS.PROGRESS_INIT; END_IF 
IF NOT Check() THEN MoveToPos   := E_PROGRESS.PROGRESS_ERROR; RETURN; END_IF


CASE _eState
OF
  E_PROGRESS.PROGRESS_INIT:
    IF Execute
    THEN
      _nErrorId               := 0;
      _rDelta                 := SEL((stMoveData.rDelta < 0.01), stMoveData.rDelta, 0.05);
      _eState                 := E_PROGRESS.PROGRESS_BUSY;
    END_IF
END_CASE
//-----------------------------------------------------------------------------
//-----------------------------------------------------------------------------
CASE _eState
OF
  E_PROGRESS.PROGRESS_BUSY:
    _eState                   := E_PROGRESS.PROGRESS_PREPARE;
    _fbPower.Override         := stMoveData.rOverride;

    _rPos                     := ABS(_Mover.NcToPlc.ModuloActTurns)* _RailLength + stMoveData.rPos;


    _rLastPosition            := _rPos;
    //_rLastGap                 := stMoveData.rGap;

    _fbMoveAbs(
            Axis              := _Mover, 
            Execute           := FALSE, 
            Position          := _rPos, 
            Velocity          := stMoveData.rVelo, 
            Acceleration      := stMoveData.rAcc, 
            Deceleration      := stMoveData.rAcc, 
            Jerk              := stMoveData.rJerk, 
            BufferMode        := Tc2_MC2.MC_BufferMode.MC_Aborting);

      IF (_eMessageLevel > E_MessageType.eMessageInfo)
      THEN
        _stMsg.eType          := E_MessageType.eMessageVerbose;
        _stMsg.eSubdevice     := e_Subdevice.fbMovePtP;
        _stMsg.iErrorNumber   := _nErrorId;
        _stMsg.sText          := concat(TO_STRING(_eState), ': ');
        _stMsg.sText          := concat(_stMsg.sText, concat('stMoveData.rPos: ', TO_STRING(stMoveData.rPos)));
        f_MessageSet(_stMsg);
      END_IF
END_CASE
//-----------------------------------------------------------------------------
//-----------------------------------------------------------------------------
CASE _eState
OF
  E_PROGRESS.PROGRESS_PREPARE:
    _fbMoveAbs(
            Axis              := _Mover, 
            Execute           := TRUE, 
            Position          := _rPos, 
            Velocity          := stMoveData.rVelo, 
            Acceleration      := stMoveData.rAcc, 
            Deceleration      := stMoveData.rAcc, 
            Jerk              := stMoveData.rJerk, 
            BufferMode        := Tc2_MC2.MC_BufferMode.MC_Aborting);

    IF _fbMoveAbs.Error
    THEN
      _bError                 := TRUE;
      _nErrorId               := _fbMoveAbs.ErrorId;
      _eState                 := E_PROGRESS.PROGRESS_ERROR;

      _stMsg.eType            := E_MessageType.eMessageError;
      _stMsg.eSubdevice       := e_Subdevice.fbMovePtP;
      _stMsg.iErrorNumber     := _nErrorId;
      _stMsg.sText            := TO_STRING(_eState);
      f_MessageSet(_stMsg);

    ELSIF _fbMoveAbs.Active OR 
          _fbMoveAbs.Done
		THEN
      _eState                 := E_PROGRESS.PROGRESS_WORKING;

      IF (_eMessageLevel = E_MessageType.eMessageVerbose)
      THEN
        _stMsg.eType          := E_MessageType.eMessageVerbose;
        _stMsg.eSubdevice     := e_Subdevice.fbMovePtP;
        _stMsg.iErrorNumber   := _nErrorId;
        _stMsg.sText          := concat(TO_STRING(_eState), ': ');
        _stMsg.sText          := concat(_stMsg.sText, '.ModuloActPos: ');
        _stMsg.sText          := concat(_stMsg.sText, TO_STRING(_Mover.NcToPlc.ModuloActPos));
        f_MessageSet(_stMsg);
      END_IF
    END_IF
END_CASE
//-----------------------------------------------------------------------------
//-----------------------------------------------------------------------------
CASE _eState
OF
  E_PROGRESS.PROGRESS_WORKING:
    _fbMoveAbs(
          Axis                := _Mover);

    IF _fbMoveAbs.Error
    THEN
      _bError                 := TRUE;
      _nErrorId               := _fbMoveAbs.ErrorId;
      _stInfo.nErrorId        := _nErrorId;
      _eState                 := E_PROGRESS.PROGRESS_ERROR;

      _stMsg.eType            := E_MessageType.eMessageError;
      _stMsg.eSubdevice       := e_Subdevice.fbMovePtP;
      _stMsg.iErrorNumber     := _nErrorId;
      _stMsg.sText            := TO_STRING(_eState);
      f_MessageSet(_stMsg);

      _fbMoveAbs( 
            Axis              := _Mover, 
            Execute           := FALSE);


    ELSIF (_Mover.NcToPlc.ActPos > _fbMoveAbs.Position - _rDelta) AND
          (_Mover.NcToPlc.ActPos < _fbMoveAbs.Position + _rDelta)
    THEN
      IF NOT _Mover.Status.Moving
      THEN
        _eState               := E_PROGRESS.PROGRESS_DONE;

        IF (_eMessageLevel > E_MessageType.eMessageError)
        THEN
          _stMsg.eType        := E_MessageType.eMessageInfo;
          _stMsg.eSubdevice   := e_Subdevice.fbMovePtP;
          _stMsg.iErrorNumber := _nErrorId;
          _stMsg.sText        := concat(TO_STRING(_eState), ': ');
          _stMsg.sText        := concat(_stMsg.sText, concat('ModActPos: ', TO_STRING(_Mover.NcToPlc.ModuloActPos)));
          f_MessageSet(_stMsg);
        END_IF
      _fbMoveAbs( 
            Axis              := _Mover, 
            Execute           := FALSE);
      END_IF
    END_IF
END_CASE
//-----------------------------------------------------------------------------
//-----------------------------------------------------------------------------

MoveToPos                   := _eState;
END_METHOD

METHOD MoveToPosCa : E_PROGRESS
VAR_INPUT
  Execute             : BOOL;
  stMoveData          : ST_MOVE_DATA;
END_VAR
VAR_INST
  _nErrorId           : UDINT;
  _rDelta,
  _rPos               : LREAL;
  _eState             : E_PROGRESS;
END_VAR
IF NOT Execute THEN _eState  := E_PROGRESS.PROGRESS_INIT; END_IF 
IF NOT Check() THEN MoveToPosCa   := E_PROGRESS.PROGRESS_ERROR; RETURN; END_IF


CASE _eState
OF
  E_PROGRESS.PROGRESS_INIT:
    IF Execute
    THEN
      _nErrorId               := 0;
      _rDelta                 := SEL((stMoveData.rDelta < 0.01), stMoveData.rDelta, 0.05);
      _eState                 := E_PROGRESS.PROGRESS_BUSY;
    END_IF
END_CASE
//-----------------------------------------------------------------------------
//-----------------------------------------------------------------------------
CASE _eState
OF
  E_PROGRESS.PROGRESS_BUSY:
    _eState                   := E_PROGRESS.PROGRESS_PREPARE;
    _fbPower.Override         := stMoveData.rOverride;

    _rPos                     := ABS(_Mover.NcToPlc.ModuloActTurns)* _RailLength + stMoveData.rPos;


    _rLastPosition            := _rPos;
    _rLastGap                 := stMoveData.rGap;

    _fbMoveAbsCa( 
            Axis              := _Mover, 
            Execute           := FALSE, 
            ContinuousUpdate  := TRUE, 
            Position          := _rPos,
            Velocity          := stMoveData.rVelo, 
            Acceleration      := stMoveData.rAcc, 
            Deceleration      := stMoveData.rAcc, 
            Jerk              := stMoveData.rJerk, 
            Gap               := stMoveData.rGap, 
            BufferMode        := Tc3_Mc3Definitions.MC_BUFFER_MODE.mcAborting);

    IF (_eMessageLevel > E_MessageType.eMessageInfo)
    THEN
      _stMsg.eType            := E_MessageType.eMessageVerbose;
      _stMsg.eSubdevice       := e_Subdevice.fbMoveToPosCa;
      _stMsg.iErrorNumber     := _nErrorId;
      _stMsg.sText            := concat(TO_STRING(_eState), ': ');
      _stMsg.sText            := concat(_stMsg.sText, concat('stMoveData.rPos: ', TO_STRING(stMoveData.rPos)));
      f_MessageSet(_stMsg);
    END_IF
END_CASE
//-----------------------------------------------------------------------------
//-----------------------------------------------------------------------------
CASE _eState
OF
  E_PROGRESS.PROGRESS_PREPARE:
    _fbMoveAbsCa( 
            Axis              := _Mover, 
            Execute           := TRUE, 
            ContinuousUpdate  := TRUE, 
            Position          := _rPos,
            Velocity          := stMoveData.rVelo, 
            Acceleration      := stMoveData.rAcc, 
            Deceleration      := stMoveData.rAcc, 
            Jerk              := stMoveData.rJerk, 
            Gap               := stMoveData.rGap, 
            BufferMode        := Tc3_Mc3Definitions.MC_BUFFER_MODE.mcAborting);

    IF _fbMoveAbsCa.Error
    THEN
      _bError                 := TRUE;
      _nErrorId               := _fbMoveAbsCa.ErrorId;
      _stInfo.nErrorId        := _nErrorId;
      _eState                 := E_PROGRESS.PROGRESS_ERROR;

      _stMsg.eType            := E_MessageType.eMessageError;
      _stMsg.eSubdevice       := e_Subdevice.fbMoveToPosCa;
      _stMsg.iErrorNumber     := _nErrorId;
      _stMsg.sText            := TO_STRING(_eState);
      f_MessageSet(_stMsg);

    ELSIF _fbMoveAbsCa.Active OR 
          _fbMoveAbsCa.Done
		THEN
      _eState                 := E_PROGRESS.PROGRESS_WORKING;

      IF (_eMessageLevel = E_MessageType.eMessageVerbose)
      THEN
        _stMsg.eType          := E_MessageType.eMessageVerbose;
        _stMsg.eSubdevice     := e_Subdevice.fbMoveToPosCa;
        _stMsg.iErrorNumber   := _nErrorId;
        _stMsg.sText          := concat(TO_STRING(_eState), ': ');
        _stMsg.sText          := concat(_stMsg.sText, '.ModuloActPos: ');
        _stMsg.sText          := concat(_stMsg.sText, TO_STRING(_Mover.NcToPlc.ModuloActPos));
        f_MessageSet(_stMsg);
      END_IF
    END_IF
END_CASE
//-----------------------------------------------------------------------------
//-----------------------------------------------------------------------------
CASE _eState
OF
  E_PROGRESS.PROGRESS_WORKING:
    _fbMoveAbsCa(
          Axis                := _Mover);

    IF _fbMoveAbsCa.Error
    THEN
      _bError                 := TRUE;
      _nErrorId               := _fbMoveAbsCa.ErrorId;
      _stInfo.nErrorId        := _nErrorId;
      _fbMoveAbsCa( 
            Axis              := _Mover, 
            Execute           := FALSE);

      _eState                 := E_PROGRESS.PROGRESS_ERROR;

